// =============================================================================
// 段 9: 合成 PID 目标位置并限位 → 调用 El_Ctrl_FB
// rPIDCmdPos = 程引插值 + 手动偏置 + 自跟踪偏置 + AGC搜索偏置 + 安全检查偏置
// =============================================================================
Axis1Remote.rPIDCmdPos:=RealTimePosCal.rInterElPos+rStepBias+rAuToStepBias+rSearchNextStepTarget+SECURITYCHECK.el_out+rAuToStepBiasTemp;
IF Axis1Remote.rPIDCmdPos<93 THEN
	Axis1Remote.rPIDCmdPos:=93;
ELSIF Axis1Remote.rPIDCmdPos>180 THEN
	Axis1Remote.rPIDCmdPos:=180;
END_IF

Axis1_Ctrl(sLocal:=Axis1Local, sCtrl:=Axis1Remote, sStatus:=Axis1Status, sVisible:=Axis1Visible, rRealPos:=rFctPosReal_1, rPosLimK:=0.34);

                  
END_PROGRAM

FUNCTION_BLOCK LinearInter
  VAR_INPUT
    tLastTime : ULINT;  (* 上一时间 *)
    rLastPos : REAL;  (* 上一时间位置 *)
    tCurTime : ULINT;  (* 当前时间 *)
    rCurPos : REAL;  (* 当前时间位置 *)
    tTargetTime : ULINT;  (* 目标时间 *)
  END_VAR
  VAR_OUTPUT
    rTargetpos : REAL;  (* 目标时间位置 *)
  END_VAR
  VAR
    iDelCurLastTime : LREAL := 1.0;  (* 当前与上一个时间差 *)
    iDelTarCurTime : LREAL := 1.0;  (* 目标与当前时间差 *)
    rK : REAL;  (* 方位斜率 *)
  END_VAR

                    //tLastTime:=tLastTime/1000000;
//tCurTime:=tCurTime/1000000;
//tTargetTime:=tTargetTime/1000000;
iDelTarCurTime:=ULINT_TO_LREAL(tTargetTime)-ULINT_TO_LREAL(tCurTime); //x1-x
IF (tCurTime-tLastTime)<>0 THEN
	iDelCurLastTime:=ULINT_TO_LREAL(tCurTime)-ULINT_TO_LREAL(tLastTime);  //x-x0
ELSE
	iDelCurLastTime:=1.0;
END_IF

IF iDelTarCurTime<>0 THEN
	rK:=(rCurPos-rLastPos)/(iDelCurLastTime);
ELSE
	rK:=0;
END_IF
rTargetpos:=rCurPos+rK*iDelTarCurTime;  //y1 + ((y1-y0)/(x1-x0))*(x-x1)
                  
END_FUNCTION_BLOCK

FUNCTION_BLOCK three2
  VAR_INPUT
    X : ARRAY[1..5] OF LREAL;
    Y : ARRAY[1..5] OF LREAL;
    y0 : REAL := 0;
    yn : REAL := 0;  (* y0,yn表示的是S''(x0)=f''(x0)=y0，S''(xn)=f''(xn)=yn,自然边界即条件值为0 *)
  END_VAR
  VAR_OUTPUT
    M : ARRAY[1..5] OF LREAL;
    A : ARRAY[1..5, 1..5] OF LREAL;
    D : ARRAY[1..3, 1..3] OF LREAL;
    g : ARRAY[1..3] OF LREAL;
    h : ARRAY[1..4] OF LREAL;
  END_VAR
  VAR
    n : INT := 5;
    ypie : ARRAY[1..5] OF REAL;
    j : INT;
    i : INT;
    u : ARRAY[1..3] OF REAL;
    n_ : ARRAY[1..3] OF REAL;
    M_ : ARRAY[1..3] OF REAL;
    solve : solvex;
    iCounttest : INT;
    miu : ARRAY[1..4] OF REAL;
  END_VAR

                    //此函数为M值求值函数
//D,h,A,g,M输出量分别为系数矩阵D，插值宽度h，差商表A，g值,M值 
n:=5;
//A(:,1)=Y'
A[1,1]:=Y[1];A[2,1]:=Y[2];A[3,1]:=Y[3];A[4,1]:=Y[4];A[5,1]:=Y[5];

//A(:,1)=Y'
FOR j :=2 TO 5 DO
	FOR i:=j TO 5 DO
		A[i,j]:=(A[i,j-1]- A[i-1,j-1])/(X[i]-X[i-j+1]);
	END_FOR
END_FOR


FOR i:=1 TO (n-1) DO
	h[i]:=X[i+1]-X[i];
END_FOR


//h[1]:=X[2]-X[1];h[2]:=X[3]-X[2];h[3]:=X[4]-X[3];h[4]:=X[5]-X[4];



//D[1,1]:=2;D[2,2]:=2;D[3,3]:=2;

FOR i:=1 TO n-2 DO
	D[i,i]:=2; 
	IF i=1 THEN
		g[i]:=(6/(h[i+1]+h[i]))*(A[i+2,2]-A[i+1,2])-h[i]/(h[i]+h[i+1])*y0;
	ELSIF i=(n-2) THEN
		g[i]:=(6/(h[i+1]+h[i]))*(A[i+2,2]-A[i+1,2])-(1-h[i]/(h[i]+h[i+1]))*yn;
	ELSE
		g[i]:=(6/(h[i+1]+h[i]))*(A[i+2,2]-A[i+1,2]);
	END_IF
END_FOR



FOR i:=2 TO (n-2) DO
	u[i]:=h[i]/(h[i]+h[i+1]);
	n_[i-1]:=h[i]/(h[i-1]+h[i]);
	D[i-1,i]:=n_[i-1];
	D[i,i-1]:=u[i];
END_FOR


solve(M:=D,G:=g,X=>M_);
M[1]:=0;M[5]:=0;M[2]:=M_[1];M[3]:=M_[2];M[4]:=M_[3];


                  
END_FUNCTION_BLOCK

FUNCTION_BLOCK threesimple2
  VAR_INPUT
    aUTC_TIME : ARRAY[1..5] OF ULINT;  (* 用于三次样条插值的数据 *)
    aPosCmd : ARRAY[1..5] OF LREAL;  (* 用于三次样条插值的数据 *)
    y0 : REAL;
    yn : REAL;  (* y0,yn表示的是S''(x0)=f''(x0)=y0，S''(xn)=f''(xn)=yn,自然边界即条件值为0 *)
    xt : REAL;  (* 所求目标位置 *)
  END_VAR
  VAR_OUTPUT
    sout : REAL;
    nout : INT;
  END_VAR
  VAR
    Three : three2;
    X : ARRAY[1..5] OF LREAL;
    Y : ARRAY[1..5] OF LREAL;
    M : ARRAY[1..5] OF LREAL;
    A : ARRAY[1..5, 1..5] OF LREAL;
    D : ARRAY[1..3, 1..3] OF LREAL;
    g : ARRAY[1..3] OF LREAL;
    h : ARRAY[1..4] OF LREAL;
    n : INT := 5;
    p1 : ARRAY[1..4] OF REAL;
    p2 : ARRAY[1..4] OF REAL;
    p3 : ARRAY[1..4] OF REAL;
    p4 : ARRAY[1..4] OF REAL;
    i : INT;
  END_VAR

                    FOR i:=1 TO 5 DO
	X[i]:=ULINT_TO_LREAL(aUTC_TIME[i]);
	Y[i]:=aPosCmd[i];
END_FOR


Three(X:=X,Y:=Y,y0:=y0,yn:=yn,D=>D,h=>h,A=>A,g=>g,M=>M);

FOR i:=1 TO (n-1) DO
	p1[i]:=M[i]*(X[i+1]-xt)*(X[i+1]-xt)*(X[i+1]-xt)/(6*h[i]);
	p2[i]:=M[i+1]*(xt-X[i])*(xt-X[i])*(xt-X[i])/(6*h[i]);
	p3[i]:=(A[i,1]-M[i]/6*(h[i])*(h[i]))*(X[i+1]-xt)/h[i];
	p4[i]:=(A[i+1,1]-M[i+1]/6*(h[i])*(h[i]))*(xt-X[i])/h[i];
	
	
END_FOR


FOR i:=1 TO (n-1) DO
	IF (xt<=X[i+1])AND (xt>=X[i]) THEN
		nout:=i;
		sout:=p1[nout]+p2[nout]+p3[nout]+p4[nout]; 
	ELSIF xt>X[5] THEN
		nout:=4;
	ELSIF xt<X[1]THEN
		nout:=1;
	END_IF
END_FOR


//要不要判断插值模块是否有效？
sout:=p1[nout]+p2[nout]+p3[nout]+p4[nout]; 
(*
IF xt>X[5] THEN
	nout:=4;
	sout:=p1[nout]+p2[nout]+p3[nout]+p4[nout]; 
ELSIF xt<X[1] THEN
	nout:=1;
	sout:=p1[nout]+p2[nout]+p3[nout]+p4[nout]; 
END_IF
*)
                  
END_FUNCTION_BLOCK

FUNCTION_BLOCK InterDataProcess
  VAR_INPUT
    ulRealTime : ULINT;  (* 实际时间 单位纳秒 *)
    Arr : ARRAY[1..5] OF ULINT := [9, 0, 1, 5, 4];  (* 创建一个包含5个整数的数组 轨道时间数组 起点 1970-01-01 0:00:00 单位纳秒 *)
  END_VAR
  VAR_OUTPUT
    MaxVal : ULINT;  (* 定义最大值、最小值和循环计数器变量 *)
    MinVal : ULINT;  (* 定义最大值、最小值和循环计数器变量 *)
    MaxIndex : INT;  (* 定义最大值和最小值的索引 *)
    MinIndex : INT;  (* 定义最大值和最小值的索引 *)
    ulInterRealTime : ULINT;  (* 插值使用的时间 *)
  END_VAR
  VAR
    i : INT;
    j : INT;
  END_VAR

                    //该功能块查找到轨道时间数组内最大最小值以及索引位置
//找出最大最小值
MaxVal := 0; // 初始化最大值
MinVal := 0; // 初始化最小值
MaxIndex := 0; // 初始化最大值的索引
MinIndex := 0; // 初始化最小值的索引

FOR i := 1 TO 5 DO
    IF Arr[i] <> 0 THEN
        IF MaxVal = 0 THEN
            MaxVal := Arr[i];
            MaxIndex := i;
        ELSIF Arr[i] > MaxVal THEN
            MaxVal := Arr[i];
            MaxIndex := i;
        END_IF

        IF MinVal = 0 THEN
            MinVal := Arr[i];
            MinIndex := i;
        ELSIF Arr[i] < MinVal THEN
            MinVal := Arr[i];
            MinIndex := i;
        END_IF
    END_IF
END_FOR

// MaxVal 和 MinVal 包含了最大值和最小值，不考虑值为0的元素
// MaxIndex 和 MinIndex 包含了最大值和最小值的索引


//当前时间和最大最小比较 
IF ulRealTime<MinVal*1000000 THEN //小于插值范围 取最小时间
	//
	ulInterRealTime:=MinVal*1000000; //应该修改插值位置 而不是时间
ELSIF ulRealTime>MaxVal*1000000THEN //大于插值范围 取最大时间
	//
	ulInterRealTime:=MaxVal*1000000;//应该修改插值位置 而不是时间
ELSE
	//如果内部有0 则不插值选取最新的数据
	FOR j:=1 TO 5 DO
		IF (Arr[i]=0) AND (j<5) THEN
			ulInterRealTime:=Arr[5];//应该修改插值位置 而不是时间
			MaxIndex:=5;
			EXIT;
		ELSIF (Arr[i]=0) AND (j=5) THEN
			//没有输入数据 需要报错吗？
		END_IF
	END_FOR
	//
END_IF
                  
END_FUNCTION_BLOCK

FUNCTION_BLOCK threesimple2_1
  VAR_INPUT
    XModbusUL : ARRAY[1..10] OF ULINT := [1, 2, 3, 4, 5, 6, 7, 8, 9, 10];  (* 输入的Modbus时间数组 *)
    XModbus : ARRAY[1..10] OF LREAL;
    YModbus : ARRAY[1..10] OF LREAL;  (* 输入的Modbus位置数组 *)
    y0 : REAL;
    yn : REAL;  (* y0,yn表示的是S''(x0)=f''(x0)=y0，S''(xn)=f''(xn)=yn,自然边界即条件值为0 *)
    xt : LREAL;  (* 所求目标位置 *)
  END_VAR
  VAR_OUTPUT
    sout : REAL;
    nout : INT;
    ErrCode : INT;
    bSetZero : BOOL;  (* Modbus序列清零标识符； *)
  END_VAR
  VAR
    Three : three2;
    X : ARRAY[1..5] OF LREAL;
    Y : ARRAY[1..5] OF LREAL;
    M : ARRAY[1..5] OF LREAL;
    A : ARRAY[1..5, 1..5] OF LREAL;
    D : ARRAY[1..3, 1..3] OF LREAL;
    g : ARRAY[1..3] OF LREAL;
    h : ARRAY[1..4] OF LREAL;
    n : INT := 5;
    p1 : ARRAY[1..4] OF REAL;
    p2 : ARRAY[1..4] OF REAL;
    p3 : ARRAY[1..4] OF REAL;
    p4 : ARRAY[1..4] OF REAL;
    i : INT;
    ii : INT;  (* 清空序列 *)
    j : INT;  (* 寻找差值区间的循环变量 *)
    k : INT;  (* 插值区间 *)
    iCountOutMaxRange : INT;
    iCountOutMinRange : INT;
    nn : INT;  (* 格式转换循环遍历 *)
    mm : INT;  (* 查重遍历； *)
  END_VAR

                    FOR nn:=1 TO 10 DO
	//XModbus[nn]:=ULINT_TO_LREAL(XModbusUL[nn])*1000000/1000.0;
	XModbus[nn]:=ULINT_TO_LREAL(XModbusUL[nn]-XModbusUL[1])+1.0;
END_FOR
	xt:=xt-ULINT_TO_LREAL(XModbusUL[1])+1.0;
IF ErrCode>0 THEN
	ErrCode:=0;
END_IF


FOR mm:=2 TO 8 DO
	IF XModbus[mm] = XModbus[mm + 1] THEN
		// 找到相等的两个数，进行线性插值
		XModbus[mm + 1] := (XModbus[mm] + XModbus[mm + 2]) / 2.0;
	END_IF;
END_FOR
IF XModbus[1] = XModbus[2] THEN
	// 找到相等的两个数，进行线性插值
	XModbus[1] := XModbus[2]-(XModbus[3]-XModbus[2]);
END_IF;
IF XModbus[9] = XModbus[10] THEN
	// 找到相等的两个数，进行线性插值
	XModbus[10] := XModbus[9]+(XModbus[9]-XModbus[8]);
END_IF;

IF ErrCode <> 0 THEN
	iCountOutMaxRange:=0;
	iCountOutMinRange:=0;
END_IF


//在何处清空序列呢
//bSetZero:=FALSE; //默认不清空

IF  XModbus[10]=0 THEN
	//报错
	ErrCode:=107;//序列为空
ELSE
	IF XModbus[10]-XModbus[1]>2000000 THEN
		sout:=YModbus[10];
	ELSE
		IF xt<XModbus[1] THEN
			sout:=YModbus[1];
			//报故障 累计超时报错
			iCountOutMinRange:=iCountOutMinRange+1;
			IF iCountOutMinRange>5000 THEN
				iCountOutMaxRange:=5001;
				//ErrCode:=108;//偏小超时报错
			END_IF
		ELSIF xt>XModbus[10]  THEN
			sout:=YModbus[10];
			//报故障 累计超时报错
			iCountOutMaxRange:=iCountOutMaxRange+1;
			IF iCountOutMaxRange>5000 THEN
				iCountOutMaxRange:=5001;
				//ErrCode:=109;//偏大超时报错
			END_IF
		ELSE //若所求目标位置在Modbus中间
			iCountOutMaxRange:=0;
			iCountOutMinRange:=0;
			//若不满五个点
			IF XModbus[6]=0 THEN
				sout:=XModbus[10];
			ELSE
				//若满五个点
				//寻找当前插值区间
				FOR j:=2 TO 10 DO
					IF xt<XModbus[j] THEN
						k:=j;
						EXIT;
					END_IF
				END_FOR
				
				IF k=2 THEN
					X[1]:=XModbus[k-1];X[2]:=XModbus[k];X[3]:=XModbus[k+1];X[4]:=XModbus[k+2];X[5]:=XModbus[k+3];
					y[1]:=YModbus[k-1];Y[2]:=YModbus[k];Y[3]:=YModbus[k+1];Y[4]:=YModbus[k+2];Y[5]:=YModbus[k+3];
				ELSIF k>2 AND k<=8 THEN
					X[1]:=XModbus[k-2];X[2]:=XModbus[k-1];X[3]:=XModbus[k];X[4]:=XModbus[k+1];X[5]:=XModbus[k+2];
					Y[1]:=YModbus[k-2];Y[2]:=YModbus[k-1];Y[3]:=YModbus[k];Y[4]:=YModbus[k+1];Y[5]:=YModbus[k+2];
				ELSIF k=9 THEN
					X[1]:=XModbus[k-3];X[2]:=XModbus[k-2];X[3]:=XModbus[k-1];X[4]:=XModbus[k];X[5]:=XModbus[k+1];
					Y[1]:=YModbus[k-3];Y[2]:=YModbus[k-2];Y[3]:=YModbus[k-1];Y[4]:=YModbus[k];Y[5]:=YModbus[k+1];
				ELSIF k=10 THEN
					X[1]:=XModbus[k-4];X[2]:=XModbus[k-3];X[3]:=XModbus[k-2];X[4]:=XModbus[k-1];X[5]:=XModbus[k];
					Y[1]:=YModbus[k-4];Y[2]:=YModbus[k-3];Y[3]:=YModbus[k-2];Y[4]:=YModbus[k-1];Y[5]:=YModbus[k];
				END_IF
				
				
				//开始解算
				Three(X:=X,Y:=Y,y0:=y0,yn:=yn,D=>D,h=>h,A=>A,g=>g,M=>M);
				FOR i:=1 TO (n-1) DO
					p1[i]:=M[i]*(X[i+1]-xt)*(X[i+1]-xt)*(X[i+1]-xt)/(6*h[i]);
					p2[i]:=M[i+1]*(xt-X[i])*(xt-X[i])*(xt-X[i])/(6*h[i]);
					p3[i]:=(A[i,1]-M[i]/6*(h[i])*(h[i]))*(X[i+1]-xt)/h[i];
					p4[i]:=(A[i+1,1]-M[i+1]/6*(h[i])*(h[i]))*(xt-X[i])/h[i];
				END_FOR
				FOR i:=1 TO (n-1) DO
					IF (xt<=X[i+1])AND (xt>=X[i]) THEN
						nout:=i;
						sout:=p1[nout]+p2[nout]+p3[nout]+p4[nout]; 
					ELSIF xt>X[5] THEN
						nout:=4;
					ELSIF xt<X[1]THEN
						nout:=1;
					END_IF
				END_FOR
				sout:=p1[nout]+p2[nout]+p3[nout]+p4[nout]; 
				(*
				IF xt>X[5] THEN
					nout:=4;
					sout:=p1[nout]+p2[nout]+p3[nout]+p4[nout]; 
				ELSIF xt<X[1] THEN
					nout:=1;
					sout:=p1[nout]+p2[nout]+p3[nout]+p4[nout]; 
				END_IF
				*)
				END_IF
			END_IF
			
		END_IF

//修正输入量为长度为10的数组

END_IF	
	




                  
END_FUNCTION_BLOCK

PROGRAM SecurityCheck
  VAR
    bPrelimit_Positive_1 : BOOL;  (* 俯仰预限位-正侧触发（上报 Modbus DI1 B15） *)
    bPrelimit_Negative_1 : BOOL;  (* 俯仰预限位-负侧触发（DI1 B13） *)
    bPrelimit_Positive_2 : BOOL;  (* 方位预限位-正侧（DI1 B11） *)
    bPrelimit_Negative_2 : BOOL;  (* 方位预限位-负侧（DI1 B09） *)
    bPrelimit_1 : BOOL;  (* 俯仰预限位硬件输入汇总（由 IO 映射赋值） *)
    bPrelimit_2 : BOOL;  (* 方位预限位硬件输入汇总 *)
    bFinallimit_1 : BOOL;  (* 俯仰终限位（DI1 B14/B12） *)
    bFinallimit_2 : BOOL;  (* 方位终限位（DI1 B10/B08） *)
    AzError : REAL;  (* 方位跟踪误差 (deg)，供扫描 FB *)
    ElError : REAL;  (* 俯仰跟踪误差 (deg)，供扫描 FB *)
    rELCurrent : REAL;  (* 俯仰伺服电流 (A 或标幺，由驱动换算) *)
    rAzCurrent : REAL;  (* 方位伺服电流 *)
    rTlCurrent : REAL;  (* 倾斜伺服电流 *)
    rAz_realpos : REAL;  (* 方位“安全逻辑用”位置 = -rFctPosReal_2 *)
    rEL_realpos : REAL;  (* 俯仰相对水平仰角 = rFctPosReal_1 - 90 *)
    fbScan : SpiralScan;  (* 直线/栅格扫描（PersistentVars.bSearchType=FALSE） *)
    fbScan1 : SpiralScan_1;  (* 螺旋扫描（bSearchType=TRUE） *)
    fbScantest : SpiralScan;  (* 测试用（已注释） *)
    enabletest : BOOL;
    aztest : REAL;  (* 测试扫描输出（非搜索时叠加到 rPosCmd） *)
    eltest : REAL;
    enable : BOOL;  (* 扫描 FB 使能：双轴程引且 AGC 达门限且未在跟踪 *)
    delta : REAL;
    n_steps : REAL;
    agc_sim : REAL;
    lock_sim : BOOL;
    cycle_cnt : INT;
    sim_done : BOOL;
    az_out : REAL;  (* 扫描给出的方位修正量 → Az rPIDCmdPos 减去此项 *)
    el_out : REAL;  (* 扫描给出的俯仰修正量 → El rPIDCmdPos 加上此项 *)
    done_out : BOOL;  (* 本轮扫描步完成 *)
    bLockSearch : BOOL;  (* 已锁定（信噪/AGC/误差电压条件满足） *)
    rSearchThre : REAL;
    rSearchThreTemp : REAL;
    bStartTrackTemp : BOOL;  (* ACU 请求自跟踪的边沿锁存 *)
    RiseEdge : R_TRIG;  (* Modbus_Slave.bStartTrackAcu 上升沿 *)
    icountLostLocking : INT;  (* 失锁计数（bType_out 路径，约 1000 拍≈10s） *)
    bErrorLock : BOOL;  (* 误差电压小于门限视为“可跟踪” *)
    icountLostLocking1 : INT;  (* 失锁计数（非 bType_out 路径，约 300 拍） *)
    bType_out : BOOL;  (* 扫描 FB 输出：扫描类型/阶段标志 *)
    iconutwait : INT;  (* 扫描完成后等待计数（用于延迟开跟踪） *)
    rdelta : REAL;  (* 螺旋扫描半径步长 *)
    rStep : REAL;  (* 螺旋扫描步数参数 *)
    bFinish : BOOL;  (* 扫描修正后误差足够小（|AzError+az_out|等） *)
    rAzErrorReal : REAL;  (* 滤波误差（已注释） *)
    rElErrorReal : REAL;
    rAlpha : REAL;  (* 滤波系数（已注释） *)
  END_VAR

                    (*==============================================================================
  PRG: SecurityCheck（远控汇总 / 安全联锁 / 捕获扫描 / 自跟踪启停）
  任务: Canopen 10ms（与 *_ctrl_1 同周期，先于或并行执行需注意调用顺序）

  主要职责:
    1. Modbus_Slave → Axis1/2/3Remote 远控命令统一赋值（阶段5 中 *_ctrl_1 注释块已移至此）
    2. 伺服电流监测（%IW10/20/30 × %ID4/9/14）
    3. 俯仰/方位跟踪误差 AzError、ElError（供螺旋/直线扫描 FB）
    4. 预限位 → GVL.Error_code 201/202，状态上报 Modbus DI1
    5. 捕获扫描 SpiralScan：输出 az_out / el_out → 叠加到 rPIDCmdPos
    6. 根据 AGC/锁相/扫描完成 自动置位 GVL.bStartTrack

  与 *_ctrl_1 关系:
    El:  rPIDCmdPos += SecurityCheck.el_out
    Az:  rPIDCmdPos -= SecurityCheck.az_out
==============================================================================*)

// =============================================================================
// 段 1: 安全逻辑用位置（与显示用 rFctPosReal 可能差符号/零点）
// =============================================================================
rAz_realpos := -1 * GVL.rFctPosReal_2;
rEl_realpos := GVL.rFctPosReal_1 - 90;

// =============================================================================
// 段 2: 三轴伺服电流监测（仅使能时读 AD，%IW×%ID/1e6）
// %IW10/%ID4=俯仰, %IW20/%ID9=方位, %IW30/%ID14=倾斜
// =============================================================================
IF Axis1Status.bServo_Enable THEN
	rELCurrent:=DINT_TO_REAL((INT_TO_DINT(%IW10)* %ID4))/1000000.0;  //俯仰轴电流监测
ELSE
	rELCurrent:=0;
END_IF

IF Axis2Status.bServo_Enable THEN
	rAzCurrent:=DINT_TO_REAL((INT_TO_DINT(%IW20)* %ID9))/1000000.0;  //方位轴电流监测
ELSE
	rAzCurrent:=0;
END_IF

IF Axis3Status.bServo_Enable THEN
	rTlCurrent:=DINT_TO_REAL((INT_TO_DINT(%IW30)* %ID14))/1000000.0;  //倾斜轴电流监测
ELSE
	rTlCurrent:=0;
END_IF

// =============================================================================
// 段 3: 跟踪误差（供 SpiralScan 判断扫描方向与完成度）
// mode2 指向: 命令位置 vs 实际位置
// mode4 程引: 插值目标+偏置 vs 实际位置（含手动/自跟踪偏置）
// =============================================================================
IF Axis2Remote.iMode = 2 THEN
	AzError:=(-1) * (Axis2Remote.rPosCmd-rFctPosReal_2);
	ElError:=Axis1Remote.rPosCmd-rFctPosReal_1;	
END_IF

IF Axis2Remote.iMode = 4 THEN
	AzError:=rFctPosReal_2-RealTimePosCal.rInterazPos-(az_ctrl_1.rStepBias+az_ctrl_1.rAuToStepBias);
	ElError:=RealTimePosCal.rInterElPos-rFctPosReal_1+ (El_ctrl_1.rStepBias+EL_ctrl_1.rAuToStepBias);
END_IF
(*
rAzErrorReal := rAzErrorReal + rAlpha * (AzError - rAzErrorReal);
rElErrorReal := rElErrorReal + rAlpha * (ElError - rElErrorReal);
*)

// =============================================================================
// 段 4: 远控故障复位（Modbus bCommReset → GVL.bError_Reset）
// =============================================================================
IF NOT GVL.bLocalCtrl THEN
	IF Modbus_Slave.bCommReset THEN
		GVL.bError_Reset:=TRUE;
	ELSE
		GVL.bError_Reset:=FALSE;
	END_IF
END_IF

// =============================================================================
// 段 5: 远控 rPosCmd 赋值（含 AGC 搜索偏置或测试扫描偏置）
// 非 bSearch: Modbus 目标 + eltest/aztest
// bSearch:   Modbus 目标 + *_ctrl_1 的 rSearchNextStepTarget_tb
// =============================================================================
IF NOT modbus_slave.bSearch THEN
	Axis1Remote.rPosCmd:=Modbus_Slave.rPosCmd_1 + eltest;
	Axis2Remote.rPosCmd:=Modbus_Slave.rPosCmd_2 - aztest;
ELSE
	Axis1Remote.rPosCmd:=Modbus_Slave.rPosCmd_1 + El_ctrl_1.rSearchNextStepTarget_tb;
	Axis2Remote.rPosCmd:=Modbus_Slave.rPosCmd_2 + Az_ctrl_1.rSearchNextStepTarget_tb;
END_IF

// =============================================================================
// 段 6: 远控三轴命令参量 — Modbus_Slave → AxisXRemote（核心汇总）
// 俯仰/方位 rPosCmd 已在段 5 赋值；此处写 mode/速度/PID/加减速等
// =============================================================================
Axis1Remote.iMode:=Modbus_Slave.iMode_1;
Axis1Remote.rVelCmd:=Modbus_Slave.rVelcmd_1;
//Axis1Remote.rPosCmd:=Modbus_Slave.rPosCmd_1;
Axis1Remote.rP:=Modbus_Slave.rP_1;
Axis1Remote.rI:=Modbus_Slave.rI_1;
Axis1Remote.rD:=Modbus_Slave.rD_1;
Axis1Remote.rPIDThre:=Modbus_Slave.rThreshold_1;
Axis1Remote.rAcceleration:=Modbus_Slave.rAcceleration_1;
Axis1Remote.rDeceleration:=Modbus_Slave.rDeceleration_1;
Axis1Remote.rVel_Limit:=Modbus_Slave.rVelLim_1;

Axis2Remote.iMode:=Modbus_Slave.iMode_2;
Axis2Remote.rVelCmd:=Modbus_Slave.rVelcmd_2;
//Axis2Remote.rPosCmd:=Modbus_Slave.rPosCmd_2;
Axis2Remote.rP:=Modbus_Slave.rP_2;
Axis2Remote.rI:=Modbus_Slave.rI_2;
Axis2Remote.rD:=Modbus_Slave.rD_2;
Axis2Remote.rPIDThre:=Modbus_Slave.rThreshold_2;
Axis2Remote.rAcceleration:=Modbus_Slave.rAcceleration_2;
Axis2Remote.rDeceleration:=Modbus_Slave.rDeceleration_2;
Axis2Remote.rVel_Limit:=Modbus_Slave.rVelLim_2;

Axis3Remote.iMode:=Modbus_Slave.iMode_3;
Axis3Remote.rVelCmd:=Modbus_Slave.rVelcmd_3;
Axis3Remote.rPosCmd:=Modbus_Slave.rPosCmd_3;
Axis3Remote.rP:=Modbus_Slave.rP_3;
Axis3Remote.rI:=Modbus_Slave.rI_3;
Axis3Remote.rD:=Modbus_Slave.rD_3;
Axis3Remote.rPIDThre:=Modbus_Slave.rThreshold_3;
Axis3Remote.rAcceleration:=Modbus_Slave.rAcceleration_3;
Axis3Remote.rDeceleration:=Modbus_Slave.rDeceleration_3;

(* 本控 HMI 赋值块已注释，本控参数由其他 POU 写入 AxisXLocal *)

// =============================================================================
// 段 7: 俯仰预限位 → Error_code 201(正)/202(负)，置位上报标志
// bPrelimit_1 由硬件 IO 映射；触发后根据当前位置方向区分正负限位
// =============================================================================
IF bPrelimit_1 THEN
	IF rFctPosReal_1>0 THEN
		bPrelimit_Positive_1:=TRUE;
		Error_code:=201;
	ELSE
		bPrelimit_Negative_1:=TRUE;
		Error_code:=202;
	END_IF;
ELSE
	bPrelimit_Negative_1:=FALSE;
	bPrelimit_Positive_1:=FALSE;
	;
END_IF

// =============================================================================
// 段 8: 方位预限位（仅置标志，Error_code 203/204 已注释）
// =============================================================================
IF bPrelimit_2 THEN
	IF rFctPosReal_2>0 THEN
		//Error_code:=203;
		bPrelimit_Positive_2:=TRUE;;
	ELSE
		//Error_code:=204;
		bPrelimit_Negative_2:=TRUE;;
	END_IF;
ELSE
	bPrelimit_Negative_2:=FALSE;
	bPrelimit_Positive_2:=FALSE;
	;
END_IF

// =============================================================================
// 段 9: 锁定判定 — 信噪比 EB_N0≥28 或 (AGC≥门限 且 误差电压≤rErrorThre)
// bErrorLock: 仅误差电压小（适合进入跟踪）
// =============================================================================
bLockSearch := READ_485.Chan1EB_N0 >= 28 OR ((GVL.Chan1AGC >= GVL.Chanthreshold) AND (SQRT(GVL.Chan1Ua * GVL.Chan1Ua + GVL.Chan1Ue * GVL.Chan1Ue) <= PersistentVars.rErrorThre));
bErrorLock  := (SQRT(GVL.Chan1Ua * GVL.Chan1Ua + GVL.Chan1Ue * GVL.Chan1Ue) <= PersistentVars.rErrorThre);

// =============================================================================
// 段 10: 捕获扫描使能 — 双轴均为程引(4)、AGC 达标或接收机锁定、且尚未自跟踪
// =============================================================================
IF Axis1Remote.iMode = 4 AND Axis2Remote.iMode = 4 AND (gvl.Chan1AGC > PersistentVars.rStartThre OR READ_485.recBuf[1] = 1) AND NOT GVL.bStartTrack THEN
	enable := TRUE;
ELSIF Axis1Remote.iMode <> 4 THEN
	enable := FALSE;
END_IF

// =============================================================================
// 段 11: 调用扫描 FB — 直线(SpiralScan) 或 螺旋(SpiralScan_1)
// 输出 az_out / el_out 在 *_ctrl_1 中叠加到 rPIDCmdPos
// =============================================================================
IF NOT PersistentVars.bSearchType THEN
	// ===== 调用直线扫描 =====
	fbScan(
		enable      := enable,
		delta       := PersistentVars.rAzScanRange,
		delta1      := PersistentVars.rElScanRange,
		n_steps     := PersistentVars.rStep,
		agc      := GVL.Chan1AGC,
		locked     := bLockSearch,
		AzError := AzError,
		elError := elError,
		bTrackState := GVL.bStartTrack,
		azimuth     => az_out,
		elevation   => el_out,
		done        => done_out,
		bType  =>bType_out
	);
ELSE
	// ===== 调用螺旋扫描====
	fbScan1(
		enable      := enable,
		delta       := rdelta,
		n_steps     := rStep,
		agc      := GVL.Chan1AGC,
		locked     := bLockSearch,
		AzError := AzError,
		elError := elError,
		azimuth     => az_out,
		elevation   => el_out,
		done        => done_out,
		bType  =>bType_out
	);
END_IF

// =============================================================================
// 段 12: 自跟踪启停状态机（仅双轴程引 mode4）
// 扫描完成+锁定 → 置 GVL.bStartTrack
// 失锁持续计数超阈值 → 清 GVL.bStartTrack
// PersistentVars.bTrackingMode: TRUE=自动开跟踪, FALSE=需 ACU 边沿 bStartTrackAcu
// =============================================================================
IF Axis1Remote.iMode = 4 AND Axis2Remote.iMode = 4 THEN
	bFinish := done_out AND (ABS(AzError + az_out) <= 0.08) AND (ABS(ElError + el_out) <= 0.08);//扫描到位
	// 上升沿检测
	RiseEdge(CLK := Modbus_Slave.bStartTrackAcu);
	
	IF RiseEdge.Q THEN
		bStartTrackTemp := TRUE;
	END_IF;
	
	IF PersistentVars.bTrackingMode THEN
		IF bType_out THEN
			IF done_out AND bLockSearch THEN
				GVL.bStartTrack := TRUE;
				icountLostLocking := 0;
			ELSIF done_out AND NOT (SQRT(GVL.Chan1Ua * GVL.Chan1Ua + GVL.Chan1Ue * GVL.Chan1Ue) <= PersistentVars.rErrorThre) THEN
				icountLostLocking := icountLostLocking + 1;
				IF icountLostLocking >= 1000 THEN //失锁持续5秒退出自跟踪
					icountLostLocking := 1001;
					GVL.bStartTrack := FALSE;
				END_IF
			END_IF
		ELSE
			IF done_out THEN
				iconutwait := iconutwait + 1;
			END_IF
			IF iconutwait >= 500 THEN
				Iconutwait := 501;
			END_IF
			IF iconutwait >= 100 AND bErrorLock AND (bFinish OR iconutwait >= 500) THEN
				GVL.bStartTrack := TRUE;
				icountLostLocking1 := 0;
			ELSIF iconutwait >= 100 AND NOT bErrorLock THEN
				icountLostLocking1 := icountLostLocking1 + 1;
				IF icountLostLocking1 >= 300 THEN //失锁持续5秒退出自跟踪
					icountLostLocking1 := 301;
					GVL.bStartTrack := FALSE;
				END_IF
			END_IF
		END_IF
	ELSE
		IF bType_out THEN
			IF done_out AND bLockSearch THEN
				GVL.bStartTrack := bStartTrackTemp;
				icountLostLocking := 0;
			ELSIF done_out AND NOT (SQRT(GVL.Chan1Ua * GVL.Chan1Ua + GVL.Chan1Ue * GVL.Chan1Ue) <= PersistentVars.rErrorThre) THEN
				icountLostLocking := icountLostLocking + 1;
				IF icountLostLocking >= 1000 THEN //失锁持续5秒退出自跟踪
					icountLostLocking := 1001;
					GVL.bStartTrack := FALSE;
				END_IF
			END_IF
		ELSE
			IF done_out THEN
				iconutwait := iconutwait + 1;
			END_IF
			IF iconutwait >= 500 THEN
				Iconutwait := 501;
			END_IF
			IF iconutwait >= 100 AND bErrorLock AND (bFinish OR iconutwait >= 500) THEN
				GVL.bStartTrack := bStartTrackTemp;
				icountLostLocking1 := 0;
			ELSIF iconutwait >= 100 AND NOT bErrorLock THEN
				icountLostLocking1 := icountLostLocking1 + 1;
				IF icountLostLocking1 >= 300 THEN //失锁持续5秒退出自跟踪
					icountLostLocking1 := 301;
					GVL.bStartTrack := FALSE;
				END_IF
			END_IF
		END_IF
	END_IF
ELSE
	bStartTrackTemp := FALSE;
	GVL.bStartTrack := Modbus_Slave.bStartTrackAcu;
	icountLostLocking := 0;
	icountLostLocking1 := 0;
	Iconutwait := 0;
END_IF

(* fbScantest 测试块已注释 *)

                  
END_PROGRAM

FUNCTION_BLOCK PID_1
  VAR_INPUT
    rTarget : REAL;  (* 设定值 *)
    rFeedback : REAL;  (* 反馈值 *)
    rPosLimPositive : LREAL;  (* 位置正限位 *)
    rPosLimNegative : LREAL;  (* 位置反限位 *)
    rKp : REAL;  (* 比例增益 *)
    rKi : REAL;  (* 积分增益 *)
    rKd : REAL;  (* 微分增益 *)
    iThreshold : INT;  (* 积分项开启的位置阈值 *)
    bPIDEnable : BOOL := TRUE;  (* PID使能 *)
    rVelLim : LREAL;  (* 速度限制 *)
  END_VAR
  VAR_OUTPUT
    rPIDOutput : LREAL := 0;  (* 带方向的输出速度 *)
  END_VAR
  VAR
    rLastError : LREAL := 0.0;  (* 上一次误差 *)
    rErrorNow : LREAL := 0.0;  (* 当前误差 *)
    rIntegralNew : LREAL := 0.0;  (* 积分项 *)
    rDerivativeNew : LREAL := 0.0;  (* 微分项 *)
    rDelta : LREAL;  (* 增量 *)
    rProportionNew : LREAL;
  END_VAR

                    
IF (bPIDEnable>0) THEN //如果PID使能
	IF rTarget=rFeedback THEN
		rPIDOutput:=0;	
	ELSE
	
		rErrorNow:=rTarget-rFeedback;//计算当前误差 en
		rProportionNew:=rErrorNow;//比例项
		//积分项
		IF rFeedback>rPosLimNegative AND rFeedback<rPosLimPositive THEN //若在软限位之内，工作时开启积分项
			IF (ABS(rTarget-rFeedback)<iThreshold OR iThreshold = -1) THEN//位置差小于积分阈值开始积分，或者设置阈值为-1，不启用这个控制
				rIntegralNew:= rIntegralNew+rErrorNow; //积分项
			ELSE
				rIntegralNew:=0;
			END_IF;
		ELSE //不在软限位范围内,则积分项为0
			rIntegralNew:=0;
		END_IF

		//PID输出
		rPIDOutPut:=rKp*rProportionNew+rKi*rIntegralNew;


		//PID限速
		
			IF rPIDOutput<(-rVelLim) THEN
				rPIDOutput:=-rVelLim;
			ELSIF rPIDOutput>rVelLim THEN
				rPIDOutput:=rVelLim;
			END_IF
		
		
		IF rFeedback>rPosLimPositive AND rPIDOutput>0 THEN 
			rPIDOutput:=0;
		END_IF
		IF rFeedback<rPosLimNegative AND rPIDOutput<0 THEN
			rPIDOutput:=0;
		END_IF
		
		rLastError:=rErrorNow;//将当前误差赋值给上一次误差
		
	END_IF
ELSE//非使能清零PID各项
	rProportionNew:=0.0;
	rIntegralNew:=0.0;
	rPIDOutput:=0.0;
END_IF










                  
END_FUNCTION_BLOCK

PROGRAM AutoTrackingCal
  VAR
    rChanUa : REAL;  (* 处理后方位误差 (V)，→ Az 自跟踪 *)
    rChanUe : REAL;  (* 处理后俯仰误差 (V)，→ El 自跟踪 *)
    rChanAGC : REAL;  (* 当前通道 AGC *)
    bChanLock : BOOL;  (* 通道锁定（保留） *)
    iCountATLock : INT;
    iState : INT;  (* 跟踪通道选择：1=通道1, 2=通道2 *)
    rAzSum : LREAL;  (* 方位累积拉偏 *)
    rElSum : LREAL;  (* 俯仰累积拉偏 *)
    rDirSenFac : REAL;  (* 方向灵敏度系数（除数） *)
    rCurentEl : LREAL;  (* 当前俯仰角弧度 (rFctPosReal_1-90) *)
    rk : LREAL;  (* 累积增益（用于 rAzSum/rElSum） *)
    rChanUaLocal : REAL;  (* 本控方位误差（未见赋值逻辑） *)
    rChanUeLocal : REAL;  (* 本控俯仰误差（未见赋值逻辑） *)
  END_VAR

                    

(*==============================================================================
  PRG: AutoTrackingCal（自跟踪误差电压处理）
  任务: Canopen 10ms
  输入: GVL.Chan1Ua/Ue/AGC/Lock（由 READ_485 写入）
  输出（程序内变量，供 *_ctrl_1 引用）:
    rChanUa  — 方位误差电压（已÷灵敏度、÷cos(俯仰)）
    rChanUe  — 俯仰误差电压（已÷灵敏度）
    rAzSum / rElSum — 累积拉偏量（当前未回写到 GVL）
  使用:
    El_ctrl_1: rChanUe → rChanU / rAuToStepBias
    Az_ctrl_1: -rChanUa → rChanU / rAuToStepBias
  注意:
    rDirSenFac、rk 在导出代码中未见赋值，可能来自 Modbus/HMI 或需人工确认
    rChanUaLocal / rChanUeLocal 未见赋值，本控自跟踪可能依赖未初始化值（原工程保留）
==============================================================================*)
(* 旧版按 iState 直接映射 GVL 通道，已注释 *)

//iState:=modbusSlave.Trace_Num;//跟踪支路选择
iState:=1;                             // 固定使用跟踪接收机 1

CASE iState OF 
	1://使用跟踪接收机1 且锁定标识为True
		// ----- 自跟踪使能且（锁定或 SecurityCheck 误差电压足够小）-----
		IF GVL.bStartTrack AND (GVL.Chan1Lock OR Securitycheck.bErrorLock) THEN
			// 方位：原始 Ua → ÷灵敏度 → ÷cos(El) 补偿大仰角时方位耦合
			rChanUa:=GVL.Chan1Ua;
			rChanUa:=rChanUa/rDirSenFac;
			rCurentEl:=(rFctPosReal_1-90)*3.1415926535897/180.0;
			rChanUa:=rChanUa/COS(rCurentEl);
			
			// 俯仰：原始 Ue → ÷灵敏度
			rChanUe:=GVL.Chan1Ue;
			rChanUe:=rChanUe/rDirSenFac;
			rChanAGC:=GVL.Chan1AGC;
			
			// 累积量（供扩展；当前 *_ctrl_1 主要用瞬时 rChanUa/Ue）
			rAzSum:=rAzSum+rk*rChanUa/1000.0;
			rElSum:=rElSum+rk*rChanUe/1000.0;
		ELSE
			rAzSum:=0;
			rElSum:=0;
			rChanUa:=0;
			rChanUe:=0;
		END_IF
		
	2://使用跟踪接收机2 且锁定标识为True
		rChanUa:=GVL.Chan2Ua;
		rChanUe:=GVL.Chan2Ue;
		rChanAGC:=GVL.Chan2AGC;
		
	3://锁定标识符为False
		//bChanLock:=FALSE;
END_CASE

                  
END_PROGRAM

PROGRAM Ti_ctrl_1
  VAR
    Axis3_Ctrl : Ti_Ctrl_FB;  (* 倾斜轴控制 FB *)
    bRemote2LocalStop : BOOL;
    bLocal2RemoteStop : BOOL;
    Error : INT;
    Axis3Limit_pos : REAL;  (* +190° *)
    Axis3Limit_Neg : REAL;  (* -190° *)
    bRTriger : Standard.R_TRIG;
    bFTriger : Standard.F_TRIG;
    Stop3_Count : INT;
    bStop_3 : BOOL;  (* 倾斜轴停稳标志 *)
    rPosModeStepBias : LREAL;
    rPosModeStep : LREAL;
    rStepBiasMax : LREAL;
    rStepBias : LREAL;
    rStep : LREAL;
    rAuToStepBias : LREAL;
    rAutoStep : LREAL;
    TbAutoTrigger : Standard.F_TRIG;
    RbAutoTrigger : Standard.R_TRIG;
    rAutoTrackingBiasMax : LREAL;
    rLocalInitPosModeSpeed : REAL;
    rRemoteInitPosModeSpeed : REAL;
    iCountOffAuto : INT;
    iCasePBAutoTrack : INT;
    rKAuToStepBias : LREAL;
    bVisError : BOOL;  (* 全局错误可视化 *)
  END_VAR

                    
(*==============================================================================
  PRG: Ti_ctrl_1（倾斜轴 Ti 顶层程序）
  任务: Canopen 10ms
  作用: 倾斜轴反馈、状态、远/本控切换保护，调用 Ti_Ctrl_FB
  与 El/Az 差异:
    - 无 AGC 搜索、无自跟踪拉偏（相关代码已注释）
    - 未在此程序内赋值 rPIDCmdPos（由 Modbus/其他模块写入后仅做限位）
    - 远控→本控切换时仅强制 Axis3Remote.iMode:=7（本控 mode 未同步置 7）
    - 本控上限钳位有一处写 Axis2Local（原工程保留，勿改）
  软限位: ±190°
==============================================================================*)
IF GVL.Error_code <> 0 THEN
	bVisError := TRUE;
ELSE
	bVisError := FALSE;
END_IF

(* 远控参量注释块为历史 Az 轴拷贝，倾斜轴参数由 Modbus_Slave 写入 Axis3Remote *)

// =============================================================================
// 段 1: 驱动状态 → Axis3Status
// =============================================================================
Axis3Status.Error := GVL.bTiStsBit3;
Axis3Status.ErrorID := GVL.eTiErrorcode;
Axis3Status.bServo_Enable := GVL.bTiStsBit0 AND GVL.bTiStsBit1 AND GVL.bTiStsBit2;
Axis3Status.bBrake := NOT (GVL.bTiStsBit0 AND GVL.bTiStsBit1 AND GVL.bTiStsBit2);
Axis3Status.Disabled := NOT (GVL.bTiStsBit0 AND GVL.bTiStsBit1 AND GVL.bTiStsBit2);
Axis3Remote.rSoft_limit_Negative:=-190;Axis3Remote.rSoft_limit_Postive:=190;
Axis3Local.rSoft_limit_Negative:=-190;Axis3Local.rSoft_limit_Postive:=190;

// =============================================================================
// 段 2: CANopen 反馈 → rFctVelReal_3 / rFctPosReal_3
// =============================================================================
rFctVelReal_3:=DINT_TO_REAL(diTiActVel)/524288.0*360.0;
rFctPosReal_3:=DINT_TO_REAL(diTiActPos)/524288.0*360.0;

// =============================================================================
// 段 3: rPosCmd 硬限位 ±190°
// 注意: 上限分支写的是 Axis2Local（原代码），与 Axis3Local 不一致，保持不改
// =============================================================================
Axis3Limit_pos:=190;
Axis3Limit_Neg:=-190;
IF Axis3Remote.rPosCmd>Axis3Limit_pos THEN
	Axis3Remote.rPosCmd:=190;
ELSIF Axis3Remote.rPosCmd<Axis3Limit_Neg THEN
	 Axis3Remote.rPosCmd:=-190;  
END_IF

IF Axis3Local.rPosCmd>Axis3Limit_pos THEN
	Axis2Local.rPosCmd:=190;
ELSIF Axis3Local.rPosCmd<Axis3Limit_Neg THEN
	 Axis3Local.rPosCmd:=-190;  
END_IF

// =============================================================================
// 段 4: 停稳判定 → Axis3Status.Moving
// =============================================================================
IF  ABS(rFctVelReal_3)<0.035 THEN
	Stop3_Count:=Stop3_Count+1;
	IF Stop3_Count>100 THEN
		Stop3_Count:=101;
		bStop_3:=TRUE;;
	END_IF
ELSE
	Stop3_Count:=0;
	bStop_3:=FALSE;
END_IF
Axis3Status.Moving := NOT bStop_3;

// =============================================================================
// 段 5: PID 使能（mode 2 / 4）
// =============================================================================
IF Axis3Remote.iMode=2 OR Axis3Remote.iMode=4 THEN
	Axis3Remote.bPIDEnable:=TRUE;
ELSE
	Axis3Remote.bPIDEnable:=FALSE;
END_IF

// =============================================================================
// 段 6: 远控 ↔ 本控 切换保护
// 远→本: 仅 Axis3Remote.iMode:=7（与 El/Az 双轴同步 halt 不同）
// =============================================================================
bRTriger(CLK:=GVL.bLocalCtrl);
bFTriger(CLK:=GVL.bLocalCtrl);

IF Axis3Status.bServo_Enable AND (bRTriger.Q ) THEN//如果速度不为0且本控发生切换，则减速停止标识为True
	bRemote2LocalStop:=TRUE;
END_IF
IF bRemote2LocalStop  THEN //若减速停止标识符为True 
	
	IF  bStop_3=TRUE THEN//且电机速度不为0 开始减速 减速完成后下使能，下使能完成后复位标识符复位
		Axis3Local.iMode:=0;
		Axis3Remote.iMode:=0;
		IF Axis3Status.bServo_Enable=FALSE THEN
			bRemote2LocalStop:=FALSE;
		END_IF
	ELSE
		Axis3Remote.iMode:=7;
	END_IF
END_IF

IF Axis3Status.bServo_Enable AND (bFTriger.Q ) THEN//如果速度不为0且本控发生切换，则减速停止标识为True
	bLocal2RemoteStop:=TRUE;
END_IF
IF bLocal2RemoteStop  THEN //若减速停止标识符为True 
	
	IF  bStop_3=TRUE THEN//且电机速度不为0 开始减速 减速完成后下使能，下使能完成后复位标识符复位
		Axis3Local.iMode:=0;
		Axis3Remote.iMode:=0;
		IF Axis3Status.bServo_Enable=FALSE THEN
			bLocal2RemoteStop:=FALSE;
		END_IF
	ELSE
		Axis3Remote.iMode:=7;
		Axis3Local.iMode:=7;
	END_IF
END_IF

(* 自跟踪与 rPIDCmdPos 程引合成在此轴已注释，当前仅对既有 rPIDCmdPos 做限位 *)

// =============================================================================
// 段 7: rPIDCmdPos 限位（赋值在其他 POU，如 Modbus_Slave / RealTimePosCal）
// =============================================================================
IF Axis3Remote.rPIDCmdPos<-190 THEN
	Axis3Remote.rPIDCmdPos:=-190;
ELSIF Axis3Remote.rPIDCmdPos>190 THEN
	Axis3Remote.rPIDCmdPos:=190;
END_IF

Axis3_Ctrl(sLocal:=Axis3Local, sCtrl:=Axis3Remote, sStatus:=Axis3Status, sVisible:=Axis3Visible, rRealPos:=rFctPosReal_3, rPosLimK:=0.34);

                  
END_PROGRAM

FUNCTION_BLOCK Ti_Ctrl_FB
  VAR_INPUT
    sLocal : AxisCrtlStruct;  (* 本控命令结构体 *)
    sCtrl : AxisCrtlStruct;  (* 远控命令结构体 *)
    sStatus : AxisStatus;  (* 轴状态 *)
    sVisible : AxisVisible;  (* HMI 可视化（此 FB 未直接使用） *)
    rRealPos : REAL;  (* 编码器实际位置 (deg) *)
    rPosLimK : REAL;  (* 备用限位系数 *)
  END_VAR
  VAR_OUTPUT
    logicError : INT;  (* 保留 *)
  END_VAR
  VAR
    VelPID_1 : PID;  (* positionMode / programBootMode 远控用 *)
    VelPID_2 : PID;  (* 本控 programBootMode 用 *)
    TON_0 : TON;  (* 超时 1s 强制下电计时器 *)
    bTick : BOOL;  (* stop0 超时标志 *)
    tr : BOOL;  (* 心跳恢复进行中标志 *)
    icount1 : INT;  (* 心跳恢复计数器1 *)
    icount2 : INT;  (* 心跳恢复计数器2 *)
    icount3 : INT;  (* 备用 *)
    bfin1 : BOOL;  (* 计数器1完成标志 *)
    bfin2 : BOOL;  (* 保留 *)
    istate : INT;  (* 上电状态机 *)
    icount : INT;  (* 上电步骤计数 *)
  END_VAR

                    (*==============================================================================
  FB: Ti_Ctrl_FB（倾斜轴 Tilt 控制功能块）
  与 El_Ctrl_FB / Az_Ctrl_FB 结构基本相同，主要差异:
    - 操作的 GVL 变量为 Ti 系列（diTiTargetVel / bTiCtrlBitX / eTiErrorcode 等）
    - 无 vpid1（Ti 轴不做变增益，programBootMode 远控直接用 VelPID_1）
    - positionMode 加速度为 10 deg/s²
    - positionMode bStartAutoTrack 分支注释掉（Ti 无自跟踪需求）
    - programBootMode 本控用 VelPID_2，参数直接来自 sLocal.rP/rI/rD
    - programBootMode 远控 bStartAutoTrack=TRUE 时调用 VelPID_1（非 vpid1）

  速度换算公式（通用）:
    diTiTargetVel [inc/s] = deg/s × 524288 / 360
==============================================================================*)

// =============================================================================
// 段 A: 轴停止或下电时清快速停止位 bit8
// =============================================================================
IF sStatus.Disabled OR(NOT sStatus.Moving)THEN
	bTiCtrlBit8 := FALSE;
END_IF

// =============================================================================
// 段 B: 全局错误复位
// =============================================================================
IF GVL.bError_Reset THEN
	sCtrl.iMode:=6;
	sLocal.iMode:=6;
	GVL.Error_code:=0;
END_IF
IF GVL.Error_code =0 THEN
	GVL.bError_Reset:=FALSE;
END_IF

// =============================================================================
// 段 C: CANopen 心跳超时（0x8130）自动恢复序列
// =============================================================================
IF GVL.eTiErrorcode = 16#8130 AND NOT tr THEN
	GVL.bTiCtrlBit7 := TRUE;
	tr:=TRUE;
	istate:=0;
	icount:=0;
	// 写入下电控制字
	GVL.bTiCtrlBit3 := FALSE;
	GVL.bTiCtrlBit0 := FALSE;
	GVL.bTiCtrlBit1 := FALSE;
	GVL.bTiCtrlBit2 := FALSE;
END_IF
IF tr THEN
	icount1 := icount1 + 1;
END_IF
IF icount1 > 101 THEN
	icount1 := 0;
	tr := FALSE;
	GVL.bTiCtrlBit7 := FALSE;
	bfin1 := TRUE;
END_IF
IF bfin1 THEN
	icount2 := icount2 + 1;
END_IF
IF icount2 > 101 THEN
	bfin1 := FALSE;
	icount2 := 0;
END_IF

// =============================================================================
// 段 D: 主控制逻辑
// =============================================================================
IF GVL.Error_code=0 AND GVL.eTiErrorcode = 0 AND NOT GVL.bTiCtrlBit7  AND NOT tr AND NOT bfin1 AND NOT bfin2 THEN

	// =========== 远控 ===========
	IF GVL.bLocalCtrl=FALSE THEN //远控
		IF sCtrl.iMode <> 1 THEN
			istate:=0;
			icount:=0;
		END_IF
		CASE sCtrl.iMode OF

			MODES.powerOff: // 下电
				IF NOT sStatus.Disabled THEN
					IF sStatus.Moving THEN // 运动中，先停止运动
						GVL.diTiTargetVel := 0;
						bTiCtrlBit8 := TRUE;
					ELSE
						// 写入下电控制字
						GVL.bTiCtrlBit3 := FALSE;
						GVL.bTiCtrlBit0 := FALSE;
						GVL.bTiCtrlBit1 := FALSE;
						GVL.bTiCtrlBit2 := FALSE;
					END_IF
				END_IF

			MODES.powerOn:  // 上电（DS402 三步序列）
				IF sStatus.Disabled THEN
					GVL.diTiTargetVel := 0;
					IF GVL.siTiMode <> 3 THEN // 上电时模式默认为3，速度模式
						GVL.siTiMode := 3;
					END_IF
					IF siTiMode = 3 THEN
						CASE istate OF
							0:
								GVL.bTiCtrlBit1 := TRUE;
								GVL.bTiCtrlBit2 := TRUE;
								icount := icount + 1;
								IF icount = 20 THEN
									icount:=0;
									istate:=1;
								END_IF
							1:
								GVL.bTiCtrlBit0 := TRUE;
								icount := icount + 1;
								IF icount = 20 THEN
									icount:=0;
									istate:=2;
								END_IF
							2:
								GVL.bTiCtrlBit3 := TRUE;
						END_CASE
					END_IF
				ELSE
					IF sStatus.Moving THEN
						GVL.diTiTargetVel := 0;
						bTiCtrlBit8 := TRUE;
					ELSE
						bTiCtrlBit8 := FALSE;
					END_IF
				END_IF

			MODES.positionMode: // 远控指向模式（加速度 10 deg/s²，Kp=0.8）
				IF NOT sStatus.Disabled THEN
					IF sCtrl.bStartAutoTrack THEN
						// Ti 轴自跟踪分支已注释掉，实际走 ELSE
						(*
						VelPID_1(rTarget:=sCtrl.rChanU + rRealPos,
								rFeedback:=rRealPos,
								rPosLimPositive:=sCtrl.rSoft_limit_Postive,
								rPosLimNegative:=sCtrl.rSoft_limit_Negative,
								rVelLim:=sCtrl.rVel_Limit,
								rKp:=sCtrl.rP_AutoTrack,//自跟踪PI系数3,0.02
								rKi:=sCtrl.rI_AutoTrack,
								rKd:=sCtrl.rD,
								bPIDEnable:=sCtrl.bPIDEnable,
								iThreshold:= -1,
								rPIDOutput=>sCtrl.rPIDCmdVel);
*)							
					ELSE
						//PID计算速度指令
						VelPID_1(rTarget:=sCtrl.rPosCmd,
							rFeedback:=rRealPos,
							rVelLim:=sCtrl.Pos_Vel,
							rPosLimPositive:=sCtrl.rSoft_limit_Postive,
							rPosLimNegative:=sCtrl.rSoft_limit_Negative,
							rKp:=0.8,//程引PI系数地带：1,0.002  高带：3,0.02
							rKi:=0,
							rKd:=0,
							bPIDEnable:=sCtrl.bPIDEnable,
							iThreshold:=sCtrl.rPIDThre,
							rPIDOutput=>sCtrl.rPIDCmdVel);
					END_IF
					GVL.diTiTargetVel := REAL_TO_DINT(sCtrl.rPIDCmdVel * 524288 / 360);
					GVL.diTiTargetAcc := REAL_TO_UDINT(10 * 524288 / 360);   //加速度 10 deg/s²
					GVL.diTiTargetDec := REAL_TO_UDINT(10 * 524288 / 360);   //减速度
				END_IF

			MODES.velocityMode://手控速度模式-远控模式
				IF NOT sStatus.Disabled THEN
					IF ABS(sCtrl.rVelCmd) <= sCtrl.rVel_Limit THEN
						GVL.diTiTargetVel := REAL_TO_DINT(sCtrl.rVelCmd * 524288 / 360);
					ELSIF sCtrl.rVelCmd > sCtrl.rVel_Limit THEN
						GVL.diTiTargetVel := REAL_TO_DINT(sCtrl.rVel_Limit * 524288 / 360);
					ELSE
						GVL.diTiTargetVel := REAL_TO_DINT(-sCtrl.rVel_Limit * 524288 / 360);
					END_IF
					GVL.diTiTargetAcc := REAL_TO_UDINT(sCtrl.rAcceleration * 524288 / 360);   //加速度
					GVL.diTiTargetDec := REAL_TO_UDINT(sCtrl.rDeceleration * 524288 / 360);   //减速度
				END_IF

			MODES.programBootMode://PID速度模式-正常模式 程引（Ti 轴用 VelPID_1，非 vpid）
				IF NOT sStatus.Disabled THEN
					IF sCtrl.bStartAutoTrack THEN
						// 程引+自跟踪：误差电压叠加到插值位置
						VelPID_1(rTarget:=sCtrl.rChanU + rRealPos,
								rFeedback:=rRealPos,
								rPosLimPositive:=sCtrl.rSoft_limit_Postive,
								rPosLimNegative:=sCtrl.rSoft_limit_Negative,
								rVelLim:=sCtrl.rVel_Limit,
								rKp:=sCtrl.rP_AutoTrack,//自跟踪PI系数3,0.02
								rKi:=sCtrl.rI_AutoTrack,
								rKd:=sCtrl.rD,
								bPIDEnable:=sCtrl.bPIDEnable,
								iThreshold:= -1,
								rPIDOutput=>sCtrl.rPIDCmdVel);							
					ELSE
						//PID计算速度指令（参数来自 sCtrl.rP/rI/rD，由 Modbus/上位机配置）
						VelPID_1(rTarget:=sCtrl.rPIDCmdPos,
							rFeedback:=rRealPos,
							rVelLim:=sCtrl.rVel_Limit,
							rPosLimPositive:=sCtrl.rSoft_limit_Postive,
							rPosLimNegative:=sCtrl.rSoft_limit_Negative,
							rKp:=sCtrl.rP,//程引PI系数地带：1,0.002  高带：3,0.02
							rKi:=sCtrl.rI,
							rKd:=sCtrl.rD,
							bPIDEnable:=sCtrl.bPIDEnable,
							iThreshold:=sCtrl.rPIDThre,
							rPIDOutput=>sCtrl.rPIDCmdVel);
					END_IF
					GVL.diTiTargetVel := REAL_TO_DINT(sCtrl.rPIDCmdVel * 524288 / 360);
					GVL.diTiTargetAcc := REAL_TO_UDINT(sCtrl.rAcceleration * 524288 / 360);   //加速度
					GVL.diTiTargetDec := REAL_TO_UDINT(sCtrl.rDeceleration * 524288 / 360);   //减速度
				END_IF

			MODES.reset://重置
				IF NOT sStatus.Disabled THEN
					IF sStatus.Moving THEN
						GVL.diTiTargetVel := 0;
						bTiCtrlBit8 := TRUE;
					ELSE
						bTiCtrlBit8 := FALSE;
					END_IF
				END_IF

			MODES.halt://待机
				IF NOT sStatus.Disabled THEN
					IF sStatus.Moving THEN
						GVL.diTiTargetVel := 0;
						bTiCtrlBit8 := TRUE;
					ELSE
						bTiCtrlBit8 := FALSE;
					END_IF
				END_IF
			
		END_CASE

	// =========== 本控 ===========
	ELSE // 本控
		IF sLocal.iMode <> 1 THEN
			istate:=0;
			icount:=0;
		END_IF
		CASE sLocal.iMode OF

			MODES.powerOff: // 下电
				IF NOT sStatus.Disabled THEN
					IF sStatus.Moving THEN // 运动中，先停止运动
						GVL.diTiTargetVel := 0;
						bTiCtrlBit8 := TRUE;
					ELSE
						// 写入下电控制字
						GVL.bTiCtrlBit3 := FALSE;
						GVL.bTiCtrlBit0 := FALSE;
						GVL.bTiCtrlBit1 := FALSE;
						GVL.bTiCtrlBit2 := FALSE;
					END_IF
				END_IF

			MODES.powerOn:  // 上电
				IF sStatus.Disabled THEN
					GVL.diTiTargetVel := 0;
					IF GVL.siTiMode <> 3 THEN // 上电时模式默认为3，速度模式
						GVL.siTiMode := 3;
					END_IF
					IF siTiMode = 3 THEN
						CASE istate OF
							0:
								GVL.bTiCtrlBit1 := TRUE;
								GVL.bTiCtrlBit2 := TRUE;
								icount := icount + 1;
								IF icount = 20 THEN
									icount:=0;
									istate:=1;
								END_IF
							1:
								GVL.bTiCtrlBit0 := TRUE;
								icount := icount + 1;
								IF icount = 20 THEN
									icount:=0;
									istate:=2;
								END_IF
							2:
								GVL.bTiCtrlBit3 := TRUE;
						END_CASE
					END_IF
				ELSE
					IF sStatus.Moving THEN
						GVL.diTiTargetVel := 0;
						bTiCtrlBit8 := TRUE;
					ELSE
						bTiCtrlBit8 := FALSE;
					END_IF
				END_IF

			MODES.velocityMode://手控速度模式-本控模式
				IF NOT sStatus.Disabled THEN
					IF ABS(sLocal.rVelCmd) <= sLocal.rVel_Limit THEN
						GVL.diTiTargetVel := REAL_TO_DINT(sLocal.rVelCmd * 524288 / 360);
					ELSIF sLocal.rVelCmd > sLocal.rVel_Limit THEN
						GVL.diTiTargetVel := REAL_TO_DINT(sLocal.rVel_Limit * 524288 / 360);
					ELSE
						GVL.diTiTargetVel := REAL_TO_DINT(-sLocal.rVel_Limit * 524288 / 360);
					END_IF
					GVL.diTiTargetAcc := REAL_TO_UDINT(sLocal.rAcceleration * 524288 / 360);   //加速度
					GVL.diTiTargetDec := REAL_TO_UDINT(sLocal.rDeceleration * 524288 / 360);   //减速度
				END_IF

			MODES.programBootMode://本控位置模式（普通 PID，参数来自 sLocal.rP/rI/rD）
				IF NOT sStatus.Disabled THEN
					IF NOT sLocal.bPIDEnable THEN
						GVL.diTiTargetVel := 0;							
					ELSE
						//PID计算速度指令
						 VelPID_2(rTarget:=sLocal.rPosCmd,
							     rFeedback:=rRealPos,
								 rPosLimPositive:=sLocal.rSoft_limit_Postive,//软限位
								 rPosLimNegative:=sLocal.rSoft_limit_Negative,
								 rKp:=sLocal.rP,
								 rKi:=sLocal.rI,
								 rKd:=sLocal.rD,
								 iThreshold:=sLocal.rPIDThre,
								 bPIDEnable:=sLocal.bPIDEnable,
								 rVelLim:=sLocal.Pos_Vel,
								 rPIDOutput=>sLocal.rPIDCmdVel);//普通PID
					END_IF
					GVL.diTiTargetVel := REAL_TO_DINT(sLocal.rPIDCmdVel * 524288 / 360);
					GVL.diTiTargetAcc := REAL_TO_UDINT(sLocal.rAcceleration * 524288 / 360);   //加速度
					GVL.diTiTargetDec := REAL_TO_UDINT(sLocal.rDeceleration * 524288 / 360);   //减速度
				END_IF

			MODES.reset://重置
			// 是否需要
			MODES.halt://待机
				IF NOT sStatus.Disabled THEN
					IF sStatus.Moving THEN
						GVL.diTiTargetVel := 0;
						bTiCtrlBit8 := TRUE;
					ELSE
						bTiCtrlBit8 := FALSE;
					END_IF
				END_IF
			
		END_CASE
	END_IF

// =============================================================================
// 段 E: 全局错误时强制停轴，超时后强制下电
// =============================================================================
ELSIF GVL.Error_code<>0 AND GVL.eTiErrorcode = 0 AND NOT GVL.bTiCtrlBit7  AND NOT tr AND NOT bfin1 AND NOT bfin2 THEN
	// 出现错误，轴停止运动
	GVL.diTiTargetVel := 0;
	bTiCtrlBit8 := TRUE;
	TON_0(IN:=bTiCtrlBit8,PT:=T#1S,Q=>,ET=>);//判断stop0执行是否超时,若超时强制下电（手动复位）
	IF TON_0.Q THEN
		bTick:=TRUE;
	END_IF
	IF bTick AND sStatus.Moving THEN // 超时强制下电
		// 写入下电控制字
		GVL.bTiCtrlBit3 := FALSE;
		GVL.bTiCtrlBit0 := FALSE;
		GVL.bTiCtrlBit1 := FALSE;
		GVL.bTiCtrlBit2 := FALSE;
	END_IF
END_IF

                  
END_FUNCTION_BLOCK

FUNCTION_BLOCK vpid
  VAR_INPUT
    rTarget : REAL;  (* 目标位置 (deg) *)
    rFeedback : REAL;  (* 实际位置 (deg) *)
    rPosLimPositive : LREAL;  (* 软限位正限 (deg) *)
    rPosLimNegitive : LREAL;  (* 软限位负限 (deg)（注：原拼写 Negitive，勿改） *)
    rKpBase : REAL;  (* Kp 基础值（低速/低角度区） *)
    rKiBase : REAL;  (* Ki 基础值 *)
    rVelThreshold : LREAL;  (* 增益切换阈值：rElPos 超过此值开始叠加增益 *)
    rKpScale : REAL;  (* Kp 随角度的线性缩放斜率 *)
    rKiScale : REAL;  (* Ki 随角度的线性缩放斜率 *)
    iThrehold : INT;  (* 积分开启的误差阈值 (deg) *)
    bPIDEnable : BOOL;  (* PID 使能 *)
    rVelLim : LREAL;  (* 输出速度限幅 (deg/s) *)
    rKpMax : REAL;  (* Kp 上限 *)
    rKiMax : REAL;  (* Ki 上限 *)
    rElPos : REAL;  (* 当前俯仰实际角度，用于动态调整增益（GVL.rFctPosReal_1-90） *)
  END_VAR
  VAR_OUTPUT
    rPIDOutput : LREAL;  (* 不带限位检查的原始输出（内部过渡量） *)
    rPIDOutDir : LREAL;  (* 最终输出速度 (deg/s)，写 diXxTargetVel 前换算 *)
  END_VAR
  VAR
    rLastFeedback : LREAL;  (* 备用（当前版本已注释掉速度计算） *)
    rErrorNow : LREAL;  (* 当前位置误差 *)
    rIntegralNew : LREAL;  (* 积分累计 *)
    rDelta : LREAL;  (* 备用 *)
    rProportionNew : LREAL;  (* 比例项 = rErrorNow *)
    rSpeed : REAL;  (* 备用（速度自适应已注释） *)
    rKp : REAL;  (* 当前实际 Kp（动态跟踪 rKpTarget） *)
    rKi : REAL;  (* 当前实际 Ki *)
    rInterValueNow : LREAL;  (* 备用（插值速度，已注释） *)
    rInterValueLast : LREAL;  (* 备用 *)
    rStep : LREAL;  (* Kp/Ki 每拍变化步长（防止突变） *)
    rKpTarget : REAL;  (* 目标 Kp（由 rElPos 计算） *)
    rKiTarget : REAL;  (* 目标 Ki *)
  END_VAR

                    (*==============================================================================
  FB: vpid（变增益自适应 PID）
  任务: Canopen 10ms（由 El_Ctrl_FB / Az_Ctrl_FB 在 programBootMode 下调用）
  作用: 与 PID 相似，但 Kp/Ki 根据当前俯仰角（rElPos）动态调整
        俯仰角越大（天线仰角越高），摩擦力和惯量变化大，需更高增益
  与 PID 的区别:
    - 输入参数带 Kp/Ki 基础值、缩放因子、最大值
    - 内部按 rElPos > rVelThreshold 时线性增加 Kp/Ki
    - 输出走 rPIDOutDir（方向输出）而非 rPIDOutput
  来源参数: PersistentVars.rXxKpBase/rXxKiBase 等（掉电保持，可由 HMI/Modbus 标定）
==============================================================================*)

// ----- 段：PID 使能入口 -----
IF (bPIDEnable) THEN // 如果PID使能
    IF rTarget = rFeedback THEN
        rPIDOutDir := 0;    
    ELSE
        rErrorNow := rTarget - rFeedback; // 计算当前误差
        rProportionNew := rErrorNow;      // 比例项
		
		// ----- 段：根据俯仰角动态计算目标 Kp/Ki -----
		// rElPos = 当前俯仰角 - 90，即相对水平的仰角
		// 当仰角 > rVelThreshold 时，增益线性增加
		IF rElPos > rVelThreshold THEN
			rKpTarget := rKpBase + rKpScale * (rElPos - rVelThreshold);
			rKiTarget := rKiBase + rKiScale * (rElPos - rVelThreshold);
		ELSE
			rKpTarget := rKpBase;
			rKiTarget := rKiBase;
		END_IF
        // ----- 段：Kp/Ki 上限保护 -----
        IF rKpTarget > rKpMax THEN
			rKpTarget := rKpMax;
		END_IF
		IF rKiTarget > rKiMax THEN
			rKiTarget := rKiMax;
		END_IF
		
		// ----- 段：Kp/Ki 平滑追踪目标值（rStep 步进，防增益突变抖动）-----
		IF rKp<=rKpTarget THEN
			rKp:=rKp+rStep;
		ELSE
			rKp:=rKp-rStep;
		END_IF
		IF rKi<=rKiTarget THEN
			rKi:=rKi+(rKiScale/rKpScale)*rStep;
		ELSE
			rKi:=rKi-(rKiScale/rKpScale)*rStep;
		END_IF
	END_IF

        // ----- 段：条件积分（与 PID 相同逻辑）-----
        IF rFeedback > rPosLimNegitive AND rFeedback < rPosLimPositive THEN // 若在软限位之内，工作时开启积分项
            IF (ABS(rTarget - rFeedback) < iThrehold) THEN // 位置差小于积分阈值
                rIntegralNew := rIntegralNew + rErrorNow;  // 积分项
            ELSE
                rIntegralNew := rIntegralNew;  // 积分项
            END_IF;
        ELSE // 不在软限位范围内，则积分项为0
            rIntegralNew := 0;
        END_IF
        (*
        // 防止目标位置与当前位置偏差过大，导致比例项输出太大，引起震动
        IF rKp * rProportionNew > 2 THEN
            rPIDOutput := 2;
        ELSIF rKp * rProportionNew < -2 THEN
            rPIDOutput := -2;
        ELSE
            rPIDOutput := rKp * rProportionNew + rKi * rIntegralNew / 1000.0; // 由于需求积分项过小，因此积分系数在接口数据上除1000
        END_IF
        *)
		rPIDOutput := rKp * rProportionNew + rKi * rIntegralNew; // 由于需求积分项过小，因此积分系数在接口数据上除1000
        // 根据方向设置输出
        IF rPIDOutput < 0 THEN
            rPIDOutDir := rPIDOutput;
        ELSE
            rPIDOutDir := rPIDOutput;
        END_IF
        
        // ----- 段：速度限幅 -----
        IF (ABS(rPIDOutDir) > rVelLim) THEN
            IF rPIDOutDir < (-rVelLim) THEN
                rPIDOutDir := -rVelLim;
            ELSIF rPIDOutDir > rVelLim THEN
                rPIDOutDir := rVelLim;
            END_IF
        END_IF
        
        // ----- 段：超软限位时强制输出清零 -----
        IF rFeedback > rPosLimPositive AND rPIDOutDir > 0  THEN
            rPIDOutDir := 0;
        END_IF
        IF rFeedback < rPosLimNegitive AND rPIDOutDir <= 0 THEN
            rPIDOutDir := 0;
        END_IF
        
        //rLastFeedback := rFeedback; // 将当前反馈值赋值给上一次反馈值
		//rInterValueLast := rInterValueNow; // 将当前插值位置值赋值给上一次

ELSE // 非使能清零PID各项
    rProportionNew := 0.0;
    rIntegralNew := 0.0;
    rPIDOutDir := 0.0;
    rPIDOutput := 0.0;
END_IF

                  
END_FUNCTION_BLOCK

PROGRAM READ_485
  VAR
    com_init : gcan.FB_Com_Init;
    com_read : gcan.FB_Com_Read;
    com_write : gcan.FB_Com_Write;
    m_uiError : UINT;
    m_out : BOOL;
    isFirst : BOOL;
    mPort : BYTE;  (* 2 = 485 口 *)
    recSize : UINT;
    recBuf : ARRAY[0..19] OF BYTE;  (* 原始接收缓冲（对外可读 recBuf[1] 等） *)
    recData : ARRAY[0..8] OF BYTE;  (* 旧协议 0x7E 帧解析用（已注释） *)
    wAGC : WORD;
    iUa : INT;
    iUe : INT;
    iChan1DataLen : UINT;
    chan1_i : INT;
    chan1_j : INT;
    Word2Bit1 : Word2Bit;  (* AGC 高低字节 → WORD *)
    Word2Bit2 : Word2Bit;  (* Ua → INT *)
    Word2Bit3 : Word2Bit;  (* Ue → INT *)
    rUagcTemp : REAL;
    rUaTemp : REAL;
    rUeTemp : REAL;
    btest : BOOL;
    btest2 : BOOL;
    rSData : REAL;  (* 信号分量（DWORD 差） *)
    rQData : REAL;  (* 噪声分量 *)
    Dword2Bit1 : Dword2Bit;  (* recBuf[8..11] → DWORD *)
    Dword2Bit2 : Dword2Bit;  (* recBuf[12..15] → DWORD *)
    Chan1EB_N0 : REAL;  (* 等效 Eb/N0 (dB)，SecurityCheck.bLockSearch 用 *)
    bEBN0Lock : BOOL;  (* 信噪比锁定标志（与模式/失锁计数相关） *)
    icount0 : INT;  (* recBuf[1]=0 累计，>400 清 bEBN0Lock *)
  END_VAR

                    

(*==============================================================================
  PRG: READ_485（跟踪接收机 RS485 通信）
  任务: SerialCom 5ms（与 GPRMC_1 同任务，端口不同）
  硬件: GCAN 串口 mPort=2（485），19200 8N1
  作用:
    - 读跟踪接收机上报帧 → 解析 AGC、Ua、Ue、锁定、Eb/N0
    - 写入 GVL.Chan1AGC / Chan1Ua / Chan1Ue / Chan1Lock
    - 输出 Chan1EB_N0、recBuf[1]、bEBN0Lock 供 SecurityCheck / 捕获扫描
  帧布局（当前简化协议，非 0x7E 定界）:
    recBuf[1]     — 锁定标志 (1=锁定)
    recBuf[2..3]  — AGC 原始 WORD
    recBuf[4..5]  — 方位误差 Ua 原始 INT
    recBuf[6..7]  — 俯仰误差 Ue 原始 INT
    recBuf[8..15] — Eb/N0 用两路 DWORD 算信噪比
==============================================================================*)

mPort:=2;								//串口端口号设定

// ----- 首次上电：485 初始化 19200 -----
IF isFirst THEN
	com_init(
	EN_IN:=TRUE,
	xEnable:=TRUE,
	bPort:=mPort,
	uiBaudrate:=19200,
	bParity:=0,
	bDatabits:=8,
	bStopbits:=1,
	EN_OUT=>m_out,
	uiError=>m_uiError);
	isfirst:=FALSE;

ELSE
	com_read(
	EN_in:=TRUE,
	bPort:=mPort,
	p_brxdata:=ADR(recBuf),
	uiMaxsize:=20,
	EN_out=>m_out,
	uiRecSize=>recSize,
	uierror=>m_uierror);
	
	// ----- 段 1: 锁定标志 → GVL.Chan1Lock -----
	//GVL.Chan1Lock := BYTE_TO_BOOL(recBuf[1]);
	IF recBuf[1] = 1 AND GVL.Chan1AGC >= GVL.Chanthreshold THEN
		GVL.Chan1Lock := TRUE;
	ELSE
		GVL.Chan1Lock := FALSE;
	END_IF

	// ----- 段 2: 按字节拼接 WORD/INT（Word2Bit UNION）-----
	Word2Bit1.Apart_Byte[1] := recBuf[2];
	Word2Bit1.Apart_Byte[2] := recBuf[3];
	wAGC:=Word2Bit1.Apart_Word;
	
	Word2Bit2.Apart_Byte[1] := recBuf[4];
	Word2Bit2.Apart_Byte[2] := recBuf[5];
	iUa:=Word2Bit2.Apart_INT;
	
	Word2Bit3.Apart_Byte[1] := recBuf[6];
	Word2Bit3.Apart_Byte[2] := recBuf[7];
	iUe:=Word2Bit3.Apart_INT;

	// ----- 段 3: 换算为物理量并限幅后写 GVL -----
	// Ua/Ue: ±5V 满量程对应 INT±2048；AGC: 5 - (raw×5/76) 越大信号越强
	IF ABS(INT_TO_REAL(iUa) * 5 / 2048) <= 5 AND ABS(INT_TO_REAL(iUe) * 5 / 2048) <= 5 AND ABS((WORD_TO_REAL(wAGC) * 5 / 76)) <=5 THEN
		GVL.Chan1Ua := INT_TO_REAL(iUa) * 5 / 2048;
		GVL.Chan1Ue := INT_TO_REAL(iUe) * 5 / 2048;
		GVL.Chan1AGC := 5 - (WORD_TO_REAL(wAGC) * 5 / 76);
	END_IF
	
	// ----- 段 4: Eb/N0 估算（两 DWORD，字节序见 Dword2Bit 填入顺序）-----
	Dword2Bit1.Apart_Byte[3] := recBuf[8];
	Dword2Bit1.Apart_Byte[4] := recBuf[9];
	Dword2Bit1.Apart_Byte[1] := recBuf[10];
	Dword2Bit1.Apart_Byte[2] := recBuf[11];	
	
	Dword2Bit2.Apart_Byte[3] := recBuf[12];
	Dword2Bit2.Apart_Byte[4] := recBuf[13];
	Dword2Bit2.Apart_Byte[1] := recBuf[14];
	Dword2Bit2.Apart_Byte[2] := recBuf[15];	
	
	rQData:=DWORD_TO_REAL(Dword2Bit2.Apart_DWORD);
	rSData:=DWORD_TO_REAL(Dword2Bit1.Apart_DWORD)-rQData;
	
	IF rSData<>0  AND rQData<>0  THEN
		Chan1EB_N0 := 10*LOG(ABS(rSData/rQData))+3.8;
	ELSE
		Chan1EB_N0 := 0;
	END_IF
	
	// ----- 段 5: bEBN0Lock — 程引/指向且 Eb/N0≥29 或 ACU 请求自跟踪 -----
	IF ((GVL.Axis1Remote.iMode = 2 OR GVL.Axis1Remote.iMode = 4) AND Chan1EB_N0 >= 29)AND READ_485.recBuf[1] = 1 OR Modbus_Slave.bStartTrackAcu THEN
		icount0:=0;
		bEBN0Lock := TRUE;
	END_IF
	// 锁定字节为 0 时累计；超 400 拍或下电则清 bEBN0Lock
	IF ( GVL.Axis1Remote.iMode = 4 or GVL.Axis1Remote.iMode =2 ) AND recBuf[1] = 0 THEN
		icount0:=icount0+1;
	END_IF
	IF icount0 > 400 OR (GVL.Axis1Remote.iMode = 0 OR GVL.Axis1Remote.iMode = 0) THEN
		icount0 := 401;
		bEBN0Lock := FALSE;
	END_IF
END_IF

(* 旧版 0x7E 定界帧解析整段已注释 *)

                  
END_PROGRAM

FUNCTION_BLOCK Get_AZ
  VAR_INPUT
    uliRealTime : LREAL;  (* 当前时间戳，单位毫秒 *)
    lrStartTime : LREAL;  (* 任务起始时间，单位秒 *)
    rNodeTime1 : REAL;
    rNodeTime2 : REAL;
    rNodeTime3 : REAL;
    rNodeTime4 : REAL;
    rNodeTime5 : REAL;
    rEndTime : REAL;
    lrFun1 : ARRAY[0..10] OF LREAL;
    lrFun2 : ARRAY[0..10] OF LREAL;
    lrFun3 : ARRAY[0..10] OF LREAL;
    lrFun4 : ARRAY[0..10] OF LREAL;
    lrFun5 : ARRAY[0..10] OF LREAL;
    lrFun6 : ARRAY[0..10] OF LREAL;
  END_VAR
  VAR_OUTPUT
    lrFitResult : LREAL;
  END_VAR
  VAR
    rDelTime : REAL;
    rRealTime : LREAL;
  END_VAR

                    rRealTime := uliRealTime / 1000.0 - lrStartTime/1000.0;


IF rRealTime <= 0.0 THEN
	rDelTime := 0.0;
	lrFitResult := lrFun1[10];
ELSIF rRealTime <= rNodeTime1 THEN
    rDelTime := rRealTime - 0.0;
	lrFitResult := lrFun1[0] * EXPT(rDelTime,10) + lrFun1[1] * EXPT(rDelTime,9) + lrFun1[2] * EXPT(rDelTime,8) + lrFun1[3] * EXPT(rDelTime,7) + lrFun1[4] * EXPT(rDelTime,6) + lrFun1[5] * EXPT(rDelTime,5)
    + lrFun1[6] * EXPT(rDelTime,4) + lrFun1[7] * EXPT(rDelTime,3) + lrFun1[8] * EXPT(rDelTime,2) + lrFun1[9] * rDelTime + lrFun1[10];
ELSIF rRealTime <= rNodeTime2 THEN
    rDelTime := rRealTime - rNodeTime1;
    lrFitResult := lrFun2[0] * EXPT(rDelTime,10) + lrFun2[1] * EXPT(rDelTime,9) + lrFun2[2] * EXPT(rDelTime,8) + lrFun2[3] * EXPT(rDelTime,7) + lrFun2[4] * EXPT(rDelTime,6) + lrFun2[5] * EXPT(rDelTime,5)
    + lrFun2[6] * EXPT(rDelTime,4) + lrFun2[7] * EXPT(rDelTime,3) + lrFun2[8] * EXPT(rDelTime,2) + lrFun2[9] * rDelTime + lrFun2[10];
ELSIF rRealTime <= rNodeTime3 THEN
    rDelTime := rRealTime - rNodeTime2;
    lrFitResult := lrFun3[0] * EXPT(rDelTime,10) + lrFun3[1] * EXPT(rDelTime,9) + lrFun3[2] * EXPT(rDelTime,8) + lrFun3[3] * EXPT(rDelTime,7) + lrFun3[4] * EXPT(rDelTime,6) + lrFun3[5] * EXPT(rDelTime,5)
    + lrFun3[6] * EXPT(rDelTime,4) + lrFun3[7] * EXPT(rDelTime,3) + lrFun3[8] * EXPT(rDelTime,2) + lrFun3[9] * rDelTime + lrFun3[10];
ELSIF rRealTime <= rNodeTime4 THEN
    rDelTime := rRealTime - rNodeTime3;
    lrFitResult := lrFun4[0] * EXPT(rDelTime,10) + lrFun4[1] * EXPT(rDelTime,9) + lrFun4[2] * EXPT(rDelTime,8) + lrFun4[3] * EXPT(rDelTime,7) + lrFun4[4] * EXPT(rDelTime,6) + lrFun4[5] * EXPT(rDelTime,5)
    + lrFun4[6] * EXPT(rDelTime,4) + lrFun4[7] * EXPT(rDelTime,3) + lrFun4[8] * EXPT(rDelTime,2) + lrFun4[9] * rDelTime + lrFun4[10];
ELSIF rRealTime <= rNodeTime5 THEN
    rDelTime := rRealTime - rNodeTime4;
    lrFitResult := lrFun5[0] * EXPT(rDelTime,10) + lrFun5[1] * EXPT(rDelTime,9) + lrFun5[2] * EXPT(rDelTime,8) + lrFun5[3] * EXPT(rDelTime,7) + lrFun5[4] * EXPT(rDelTime,6) + lrFun5[5] * EXPT(rDelTime,5)
    + lrFun5[6] * EXPT(rDelTime,4) + lrFun5[7] * EXPT(rDelTime,3) + lrFun5[8] * EXPT(rDelTime,2) + lrFun5[9] * rDelTime + lrFun5[10];
ELSIF rRealTime <= rEndTime THEN
    rDelTime := rRealTime - rNodeTime5;
    lrFitResult := lrFun6[0] * EXPT(rDelTime,10) + lrFun6[1] * EXPT(rDelTime,9) + lrFun6[2] * EXPT(rDelTime,8) + lrFun6[3] * EXPT(rDelTime,7) + lrFun6[4] * EXPT(rDelTime,6) + lrFun6[5] * EXPT(rDelTime,5)
    + lrFun6[6] * EXPT(rDelTime,4) + lrFun6[7] * EXPT(rDelTime,3) + lrFun6[8] * EXPT(rDelTime,2) + lrFun6[9] * rDelTime + lrFun6[10];
ELSE
    rDelTime := rEndTime - rNodeTime5;
    lrFitResult := lrFun6[0] * EXPT(rDelTime,10) + lrFun6[1] * EXPT(rDelTime,9) + lrFun6[2] * EXPT(rDelTime,8) + lrFun6[3] * EXPT(rDelTime,7) + lrFun6[4] * EXPT(rDelTime,6) + lrFun6[5] * EXPT(rDelTime,5)
    + lrFun6[6] * EXPT(rDelTime,4) + lrFun6[7] * EXPT(rDelTime,3) + lrFun6[8] * EXPT(rDelTime,2) + lrFun6[9] * rDelTime + lrFun6[10];
END_IF

IF lrFitResult>270 THEN
	lrFitResult:=270;
ELSIF lrFitResult<-270 THEN
	lrFitResult:=-270;
END_IF
                  
END_FUNCTION_BLOCK

FUNCTION_BLOCK Get_AZ_1
  VAR_INPUT
    uliRealTime : LREAL;  (* 当前时间戳，单位毫秒 *)
    lrStartTime : LREAL;  (* 任务起始时间，单位秒 *)
    rNodeTime1 : REAL;
    rNodeTime2 : REAL;
    rNodeTime3 : REAL;
    rNodeTime4 : REAL;
    rNodeTime5 : REAL;
    rEndTime : REAL;
    lrFun1 : ARRAY[0..10] OF LREAL;
    lrFun2 : ARRAY[0..10] OF LREAL;
    lrFun3 : ARRAY[0..10] OF LREAL;
    lrFun4 : ARRAY[0..10] OF LREAL;
    lrFun5 : ARRAY[0..10] OF LREAL;
    lrFun6 : ARRAY[0..10] OF LREAL;
  END_VAR
  VAR_OUTPUT
    lrFitResult : LREAL;
  END_VAR
  VAR
    rDelTime : REAL;
    rRealTime : LREAL;
  END_VAR

                    rRealTime := uliRealTime / 1000.0 - lrStartTime/1000.0;


IF rRealTime <= 0.0 THEN
	rDelTime := 0.0;
	lrFitResult := lrFun1[10];
ELSIF rRealTime <= rNodeTime1 THEN
    rDelTime := rRealTime - 0.0;
	lrFitResult := lrFun1[0] * EXPT(rDelTime,10) + lrFun1[1] * EXPT(rDelTime,9) + lrFun1[2] * EXPT(rDelTime,8) + lrFun1[3] * EXPT(rDelTime,7) + lrFun1[4] * EXPT(rDelTime,6) + lrFun1[5] * EXPT(rDelTime,5)
    + lrFun1[6] * EXPT(rDelTime,4) + lrFun1[7] * EXPT(rDelTime,3) + lrFun1[8] * EXPT(rDelTime,2) + lrFun1[9] * rDelTime + lrFun1[10];
ELSIF rRealTime <= rNodeTime2 THEN
    rDelTime := rRealTime - rNodeTime1;
    lrFitResult := lrFun2[0] * EXPT(rDelTime,10) + lrFun2[1] * EXPT(rDelTime,9) + lrFun2[2] * EXPT(rDelTime,8) + lrFun2[3] * EXPT(rDelTime,7) + lrFun2[4] * EXPT(rDelTime,6) + lrFun2[5] * EXPT(rDelTime,5)
    + lrFun2[6] * EXPT(rDelTime,4) + lrFun2[7] * EXPT(rDelTime,3) + lrFun2[8] * EXPT(rDelTime,2) + lrFun2[9] * rDelTime + lrFun2[10];
ELSIF rRealTime <= rNodeTime3 THEN
    rDelTime := rRealTime - rNodeTime2;
    lrFitResult := lrFun3[0] * EXPT(rDelTime,10) + lrFun3[1] * EXPT(rDelTime,9) + lrFun3[2] * EXPT(rDelTime,8) + lrFun3[3] * EXPT(rDelTime,7) + lrFun3[4] * EXPT(rDelTime,6) + lrFun3[5] * EXPT(rDelTime,5)
    + lrFun3[6] * EXPT(rDelTime,4) + lrFun3[7] * EXPT(rDelTime,3) + lrFun3[8] * EXPT(rDelTime,2) + lrFun3[9] * rDelTime + lrFun3[10];
ELSIF rRealTime <= rNodeTime4 THEN
    rDelTime := rRealTime - rNodeTime3;
    lrFitResult := lrFun4[0] * EXPT(rDelTime,10) + lrFun4[1] * EXPT(rDelTime,9) + lrFun4[2] * EXPT(rDelTime,8) + lrFun4[3] * EXPT(rDelTime,7) + lrFun4[4] * EXPT(rDelTime,6) + lrFun4[5] * EXPT(rDelTime,5)
    + lrFun4[6] * EXPT(rDelTime,4) + lrFun4[7] * EXPT(rDelTime,3) + lrFun4[8] * EXPT(rDelTime,2) + lrFun4[9] * rDelTime + lrFun4[10];
ELSIF rRealTime <= rNodeTime5 THEN
    rDelTime := rRealTime - rNodeTime4;
    lrFitResult := lrFun5[0] * EXPT(rDelTime,10) + lrFun5[1] * EXPT(rDelTime,9) + lrFun5[2] * EXPT(rDelTime,8) + lrFun5[3] * EXPT(rDelTime,7) + lrFun5[4] * EXPT(rDelTime,6) + lrFun5[5] * EXPT(rDelTime,5)
    + lrFun5[6] * EXPT(rDelTime,4) + lrFun5[7] * EXPT(rDelTime,3) + lrFun5[8] * EXPT(rDelTime,2) + lrFun5[9] * rDelTime + lrFun5[10];
ELSIF rRealTime <= rEndTime THEN
    rDelTime := rRealTime - rNodeTime5;
    lrFitResult := lrFun6[0] * EXPT(rDelTime,10) + lrFun6[1] * EXPT(rDelTime,9) + lrFun6[2] * EXPT(rDelTime,8) + lrFun6[3] * EXPT(rDelTime,7) + lrFun6[4] * EXPT(rDelTime,6) + lrFun6[5] * EXPT(rDelTime,5)
    + lrFun6[6] * EXPT(rDelTime,4) + lrFun6[7] * EXPT(rDelTime,3) + lrFun6[8] * EXPT(rDelTime,2) + lrFun6[9] * rDelTime + lrFun6[10];
ELSE
    rDelTime := rEndTime - rNodeTime5;
    lrFitResult := lrFun6[0] * EXPT(rDelTime,10) + lrFun6[1] * EXPT(rDelTime,9) + lrFun6[2] * EXPT(rDelTime,8) + lrFun6[3] * EXPT(rDelTime,7) + lrFun6[4] * EXPT(rDelTime,6) + lrFun6[5] * EXPT(rDelTime,5)
    + lrFun6[6] * EXPT(rDelTime,4) + lrFun6[7] * EXPT(rDelTime,3) + lrFun6[8] * EXPT(rDelTime,2) + lrFun6[9] * rDelTime + lrFun6[10];
END_IF

IF lrFitResult>90 THEN
	lrFitResult:=90;
ELSIF lrFitResult<3 THEN
	lrFitResult:=3;
END_IF
                  
END_FUNCTION_BLOCK

FUNCTION_BLOCK AGCMaxSearch_PB_1
  VAR_INPUT
    bstart : BOOL;  (* 模块开始标识 *)
    rAGCNow : REAL;  (* 当前AGC值 *)
    btrig : BOOL;  (* 触发一次 *)
    rStepBiasNow : REAL;  (* 当前拉偏量 //用来判断此次搜索是否有效 *)
    bAutoTracking : BOOL;  (* 自跟踪标识 *)
    bStop : BOOL;  (* 满足ua ue很小 *)
    rCurrentPos : REAL;  (* 当前位置 *)
    rInterPos : REAL;  (* 插值位置 *)
  END_VAR
  VAR_OUTPUT
    rAGCMaxBias : REAL;  (* 输出AGC最强时的拉偏量 单位为° *)
    bSucess : BOOL;  (* 数出模块是否成功 *)
    rStepBias : REAL;  (* 步进量 *)
  END_VAR
  VAR
    ton : Standard.TON;
    rTrg : Standard.R_TRIG;  (* 初始化上升沿检测器 *)
    rAGCInit : REAL := 0;  (* 初始化AGC *)
    rPrevAGC : REAL := 0;  (* 上一步的AGC值 单位为V *)
    rBiasInit : REAL;  (* 初始化拉偏量 *)
    iCountStep : INT := 0;  (* 计步数 *)
    toN1 : Standard.Ton;  (* 计时器 定时触发上升沿 *)
    rDirection : INT := 1;
    rSearchNextStepTarget : REAL;  (* 搜索当前目标位置 单位为° *)
    rStep : REAL := 0.0003;  (* 步进值 *)
    rSensitivity : REAL := 0.05;  (* 反向灵敏度 *)
    iCountStopMax : INT := 20;  (* 停止计数上限 *)
    rLastDirection : INT;  (* 上一次方向，判断是否换向 *)
    iCountDirChange : INT;  (* 换向标识 *)
    rAGCMaxPos : REAL;  (* 信号最强位置 *)
    rAGCLastrecord : REAL;
    iStatus : INT;
    iCountStop1 : INT;  (* 第一阶段停止标识 (正向) *)
    iCountStop2 : INT;  (* (反向) *)
    rAGCMaxValue : REAL;  (* AGC最大值 *)
    iCountSearchRight : INT;  (* 搜索方向正确，提前结束标识 *)
    bSearchRight : BOOL;  (* 搜索正确标识 *)
    iCountBlockEnd : INT;  (* 用来计数确认已达到最强位置 *)
    iCountBlockEndMax : INT := 500;  (* 到位计数上限 *)
  END_VAR

                    
(*==============================================================================
  FB: AGCMaxSearch_PB_1（AGC 峰值搜索：单轴拉偏搜索）
  调用者: `Az_ctrl_1` / `El_ctrl_1`
  目标: 在指向(mode2)或程引(mode4)时，沿单轴正/负方向试探移动 rStepBias，
        找到使 AGC 最大的位置偏置 rAGCMaxBias，并在到位稳定后置 bSucess

  关键变量含义:
    rStepBias      — 当前偏置输出（逐步累加 rDirection*rStep）
    rAGCMaxBias    — 历史最大 AGC 对应的偏置
    rAGCInit       — 启动时 AGC 基线
    rSensitivity   — 判定“AGC 明显下降/上升”的阈值，用于决定停止/换向
    iCountDirChange— 换向次数；=2 后进入“回到峰值位置并等待稳定”阶段

  完成判定:
    - 偏置回到 rAGCMaxBias 后，(rInterPos+rStepBias) 与 rCurrentPos 误差持续小于 0.002
    - 持续计数超过 iCountBlockEndMax 后，再用 TON(1s) 确认稳定 → bSucess=TRUE
==============================================================================*)

rTrg(CLK:=bstart,Q=>);

IF rTrg.Q THEN
	rAGCInit:=rAGCNow;
	rAGCMaxValue:=rAGCNow;
	//rBiasInit:=rCurrentPos-rInterPos;//获取启动时的拉偏量
END_IF

IF bstart THEN
	//搜索换向两次
	IF iCountDirChange=2 THEN
		rSearchNextStepTarget:=rAGCMaxBias;
		IF rStepBias< rSearchNextStepTarget THEN 
			rStepBias:=rStepBias+rStep;
		ELSIF rStepBias> rSearchNextStepTarget THEN
			rStepBias:=rStepBias-rStep;
		ELSE
			rStepBias:=rStepBias;
		END_IF
		
		IF ABS((rInterPos+rStepBias)-rCurrentPos)<0.002 THEN //若位置达到最强位置，则输出成功 //可能只是路过这里,需要持续
			//需要判断稳定
			iCountBlockEnd:=iCountBlockEnd+1;
		ELSE
			iCountBlockEnd:=0;
		END_IF
		IF iCountBlockEnd>iCountBlockEndMax THEN
			iCountBlockEnd:=iCountBlockEndMax+1;
			//用TON1秒后触发
			ton(IN:=TRUE,PT:=T#1S,Q=>,ET=>);
		END_IF
		IF ton.Q THEN
			bSucess:=TRUE;
		END_IF
	ELSE
		rStepBias:=rStepBias+rDirection*rStep;
		IF rDirection<0 THEN
			//若是向小走
			IF rCurrentPos<rInterPos THEN
				IF rAGCNow<rAGCMaxValue-rSensitivity THEN
					iCountStop1:=iCountStop1+1;
					IF iCountStop1>iCountStopMax THEN
						iCountStop1:=iCountStopMax+1;
						IF bSearchRight THEN
							iCountDirChange:=2;
						ELSE
							iCountDirChange:=iCountDirChange+1;
						END_IF
						rDirection:=rDirection*(-1);
					END_IF
				ELSE
					iCountStop1:=0;	
				END_IF
				
				//新加的 测试第一阶段搜索正确后不进行第二次搜索
				IF rAGCNow>rAGCInit+rSensitivity THEN
					iCountSearchRight:=iCountSearchRight+1;
				ELSE
					iCountSearchRight:=0;
				END_IF
				IF iCountSearchRight>200 THEN
					iCountSearchRight:=201;
					bSearchRight:=TRUE;
				END_IF
				
			END_IF
		ELSE
			//若是向正走
			IF rCurrentPos>rInterPos THEN
				IF rAGCNow<rAGCMaxValue-rSensitivity THEN
					iCountStop2:=iCountStop2+1;
					IF iCountStop2>iCountStopMax THEN
						iCountStop2:=iCountStopMax+1;
						IF bSearchRight THEN
							iCountDirChange:=2;
						ELSE
							iCountDirChange:=iCountDirChange+1;
						END_IF
						rDirection:=rDirection*(-1);
					END_IF
				ELSE
					iCountStop2:=0;	
				END_IF
				
				//新加的
				IF rAGCNow>rAGCInit+rSensitivity THEN
					iCountSearchRight:=iCountSearchRight+1;
				ELSE
					iCountSearchRight:=0;
				END_IF
				IF iCountSearchRight>200 THEN
					iCountSearchRight:=201;
					bSearchRight:=TRUE;
				END_IF
				
			END_IF
		END_IF
		(*
		IF rAGCNow<rAGCInit-0.05 THEN
			iCountStop1:=iCountStop1+1;
			IF iCountStop1>150 THEN
				iCountDirChange:=iCountDirChange+1;
				rDirection:=rDirection*(-1);
			END_IF
		ELSE
			iCountStop1:=0;	
		END_IF
		*)
		
		 // 记录最强信号的拉偏量和值
		//IF rAGCNow >= rAGCInit AND rAGCNow> rAGCMaxValue THEN
		IF  rAGCNow> rAGCMaxValue THEN
			rAGCMaxBias := rStepBias;
			rAGCMaxValue := rAGCNow;
		END_IF
	END_IF
ELSE
	rStepBias:=0;
	//清空变量
	iCountDirChange:=0;
	rAGCInit:=0;
	rAGCMaxValue:=0;
	rAGCMaxBias:=0;
	rDirection:=1;
	iCountStop1:=0;
	iCountStop2:=0;
	ton(IN:=FALSE,PT:=T#1S,Q=>,ET=>);
	//rStepBias:=0;
	rSearchNextStepTarget:=0;
	bSucess:=FALSE;
	iCountSearchRight:=0;
	bSearchRight:=FALSE;
	iCountBlockEnd:=0;
END_IF


(*
IF rStepBias< rSearchNextStepTarget THEN 
	rStepBias:=rStepBias+rStep;
ELSIF rStepBias> rSearchNextStepTarget THEN
	rStepBias:=rStepBias-rStep;
ELSE
	rStepBias:=rStepBias;
END_IF*)
                  
END_FUNCTION_BLOCK

PROGRAM GPRMC_1
  VAR
    com_init : gcan.FB_Com_Init;  (* gcan.FB_Com_Init为串口初始化功能块，可设定串口端口号，串口波特率等参数 *)
    com_read : gcan.FB_Com_Read;  (* gcan.FB_Com_Read为串口接收功能块，用于通过接收串口发送给PLC的数据 *)
    com_write : gcan.FB_Com_Write;  (* gcan.FB_Com_Write为串口发送功能块，用于发送串口数据 *)
    m_uiError : UINT;  (* 用于承接功能块中报错引脚错误信息的变量 *)
    m_out : BOOL;  (* 用于承接功能块中完成标志引脚数据的变量 *)
    isFirst : BOOL := TRUE;  (* 用于判断初始化只执行一次的逻辑 *)
    mPort : BYTE;  (* 程序中用作设定串口端口号 *)
    recSize : UINT;  (* 接收数据长度，单位：字节 *)
    recBuf : ARRAY[0..101] OF BYTE;  (* 用于存放接收到的串口数据的数组 *)
    sum_i : INT;
    checksum : BYTE;
    iYear : INT;
    iMonth : INT;
    iDay : INT;
    iHour : INT;
    iMinute : INT;
    iSecond : INT;
    strDateTimeNow : STRING;
    gnssTimestamp : ULINT;
    gnssTimestamplast : ULINT;
    icount : INT;
    high4 : BYTE;
    low4 : BYTE;
  END_VAR
  VAR_INPUT
    EN_in_1 : BOOL;
  END_VAR

                    (*==============================================================================
  PRG: GPRMC_1（GNSS 串口接收与 NMEA 时间解析）
  任务: SerialCom 5ms
  硬件: GCAN 模块串口 mPort=1（232），115200 8N1
  作用:
    - 读 GNSS 模块输出的 NMEA 报文（GPRMC 等，帧头 ASCII '$'=36）
    - 从固定偏移解析 UTC 日期时间，+8 转为北京时间
    - 写入 GVL.stGNSS_Timestap（毫秒 ULINT），供 TimeAdd / RealTimePosCal 使用
  下游:
    TimeAdd.icount — 秒未变时累加，用于 GNSS 丢帧时的 10ms 插值
    RealTimePosCal — GVL.dRealTime := stGNSS_Timestap + 10*TimeAdd.icount
==============================================================================*)


////////////////////////////////////////////////////////////////////////////////////////
//串口接收GPRMC报文解析
//日期：2024/08/25
//版本：V1.1
/////////////////////////////////////////////////////////////////////////////////////////

mPort:=1;								//串口端口号设定，GCAN-PLC-400、GCAN-PLC-510、GCAN-PLC-511，1为232，2为485
										//GCAN-PLC-324、GCAN-PLC-326，1为第一路485，2为第2路485
IF isFirst THEN
	com_init(							//串口初始化功能块
	EN_IN:=TRUE,						//串口初始化功能块使能
	xEnable:=TRUE,						//串口功能使能
	bPort:=mPort,						//串口端口号设定
	uiBaudrate:=115200,					//串口波特率设定
	bParity:=0,							//串口奇偶校验设定，0为无校验，1为奇校验，2为偶检验
	bDatabits:=8,						//数据位设定
	bStopbits:=1,						//停止位设定
	EN_OUT=>m_out,						//串口初始化功能块执行完成标志位
	uiError=>m_uiError);				//串口初始化功能块执行错误信息
	isfirst:=FALSE;						//执行一次初始化后关闭IF的条件使其之后进入ELSE程序段运行

ELSE
	
		com_read(						//串口读取功能块
		EN_in:=TRUE,					//读取功能块使能，为TRUE执行读取
		bPort:=mPort,					//串口端口号设定
		p_brxdata:=ADR(recBuf),			//读取到的串口数据引脚为指针类型，使用ADR()指向自建数组将数据存放到数组中
		uiMaxsize:=204,					//设定最大读取长度
		EN_out=>m_out,					//串口读取功能块执行完成标志位******功能块执行完成不代表接收完成********
		uiRecSize=>recSize,				//串口接收数据长度，单位：字节，大于0时说明接收到数据可用于判断是否接收
		uierror=>m_uierror);			//串口读取功能块执行错误信息
										//从数组recBuf里取数据，解析出年、月、日、时、分、秒
		//有效判定(A)+和校验(hh),前 4bit和后 4bit的 16 进制数分别以 ASCII 码表示(0~9,A~F)，高位在前。
		IF 	recBuf[0] = 36 THEN
(*			checksum := 16#00;
			FOR sum_i:=1 TO 74 BY 1 DO
				checksum:= checksum XOR recBuf[sum_i];
			END_FOR
			high4 := (SHR(checksum, 4) AND 16#0F)+16#30;
			low4 := (checksum AND 16#0F)+16#30;
			IF recBuf[76]= high4 AND recBuf[77]= low4 THEN 
*)		

			iYear:=BYTE_TO_INT(recBuf[23]-48)*1000+BYTE_TO_INT(recBuf[24]-48)*100+BYTE_TO_INT(recBuf[25]-48)*10+BYTE_TO_INT(recBuf[26]-48);
			iMonth:=BYTE_TO_INT(recBuf[20]-48)*10+BYTE_TO_INT(recBuf[21]-48);
			iDay:=BYTE_TO_INT(recBuf[17]-48)*10+BYTE_TO_INT(recBuf[18]-48);
			iHour:=BYTE_TO_INT(recBuf[7]-48)*10+BYTE_TO_INT(recBuf[8]-48)+8;
			iMinute:=BYTE_TO_INT(recBuf[9]-48)*10+BYTE_TO_INT(recBuf[10]-48);
			iSecond:=BYTE_TO_INT(recBuf[11]-48)*10+BYTE_TO_INT(recBuf[12]-48);
			
			// 计算时间戳		
			
			strDateTimeNow := CONCAT(STR1 := 'DT#', STR2 := INT_TO_STRING(iYear));
			strDateTimeNow := CONCAT(STR1 := strDateTimeNow, STR2 := '-');
			strDateTimeNow := CONCAT(STR1 := strDateTimeNow, STR2 := INT_TO_STRING(iMonth));
			strDateTimeNow := CONCAT(STR1 := strDateTimeNow, STR2 := '-');
			strDateTimeNow := CONCAT(STR1 := strDateTimeNow, STR2 := INT_TO_STRING(iDay));
			strDateTimeNow := CONCAT(STR1 := strDateTimeNow, STR2 := '-');
			strDateTimeNow := CONCAT(STR1 := strDateTimeNow, STR2 := INT_TO_STRING(iHour));
			strDateTimeNow := CONCAT(STR1 := strDateTimeNow, STR2 := ':');
			strDateTimeNow := CONCAT(STR1 := strDateTimeNow, STR2 := INT_TO_STRING(iMinute));
			strDateTimeNow := CONCAT(STR1 := strDateTimeNow, STR2 := ':');
			strDateTimeNow := CONCAT(STR1 := strDateTimeNow, STR2 := INT_TO_STRING(iSecond));
			(*
			gnssTimestamplast:=gnssTimestamp;
			
			
			*)
			gnssTimestamp := DT_TO_ULINT(TO_DT(strDateTimeNow)) * 1000;
			GVL.stGNSS_Timestap := gnssTimestamp;
		END_IF
		(*
		IF gnssTimestamplast<>gnssTimestamp THEN
			icount:=0;
		ELSE
			icount:=icount+1;
		END_IF
		*)
		


(*	IF recsize>0 THEN					//如果接收到串口数据
		
		com_write(						//串口发送功能块
		EN_IN:=TRUE,					//串口发送功能块使能，发送机制：当使能为TRUE时，PLC程序每周期运行到此处就执行一次发送
		bPort:=mPort,					//串口端口号设定
		p_bTxdata:=ADR(recbuf),			//将接收存放到数组中的数据发送出去******若发送其它数据，自建另一数组用于存放发送数据即可
		uiTxsize:=recsize,				//发送长度为接收到的数据长度******若发送其它长度，自行填写所需长度即可
		EN_OUT=>m_out,					//串口发送功能块执行完成标志位
		uierror=>m_uierror);			//串口发送功能块执行错误信息
			
	END_IF
*)	
END_IF
                  
END_PROGRAM

PROGRAM GetACUTime
  VAR
    tp : TP;  (* 脉冲定时器 *)
    toggle : BOOL := FALSE;  (* 当前输出状态 *)
    clk : BOOL := FALSE;  (* 方波输出 *)
    tick_ms : TIME := TIME#500ms;  (* 高电平/低电平持续时间 *)
    Result : RTS_IEC_RESULT;
    stUTC_Timestamp : SYSTIME;
    dRTime : ULINT;  (* 上位机外部时间 单位ns Unix时间戳，起点是1970-1-1 0:0:0 *)
    dModbusTime : ULINT;  (* Modbus临时外部时间 *)
    iCountRemote : INT;  (* 上位机锁定判断时间常数 *)
    dCountRemote : ULINT;  (* 上位机时间滑动平均常数 *)
    dLastRTime : ULINT;  (* 上位机上一次外部时间 单位ns Unix时间戳，起点是1970-1-1 0:0:0 *)
    iDiffRTime : DINT;  (* 上位机时间差值 *)
    dDelRTime : LINT;
    dMeanDelRTime : LINT;
    rTriger : Standard.R_TRIG;  (* 上升沿触发器 *)
    iDiff : DINT;  (* 实际时间差值 *)
    iDiffLocal : DINT;  (* 本地时间差值 *)
    iDiffETime : DINT;  (* 外部时间差值 *)
    ulACUTimeStamp : ULINT;
  END_VAR

                    
// 每次TP结束时翻转状态
IF NOT tp.Q THEN
    toggle := NOT toggle;
    tp.IN := TRUE;
    tp.PT := tick_ms;
ELSE
    tp.IN := FALSE;
END_IF

tp();

Result := SysTimeRtcHighResGet(stUTC_Timestamp);
rTriger(CLK:=toggle);
IF rTriger.Q THEN
	dRTime := modbus_slave.UTC_New;
	iDiffRTime:=ULINT_TO_DINT(dRTime-dLastRTime);
	IF ABS(iDiffRTime)>500 THEN //两次PTP时间差如果大于500毫秒,则判断为上位机时间失锁
		iCountRemote:=0;
		dCountRemote:=0;
		GVL.bRemoteTimeLock:=FALSE;
	ELSE//否则判断为上位机时间锁定并累计1分钟
		iCountRemote:=iCountRemote+1;
	END_IF
	
	IF iCountRemote>=20 THEN //累计20s认为时间可用
		iCountRemote:=20;
		dDelRTime := TO_ULINT(stUTC_Timestamp) - (dRTime + 8 * 3600 *1000);
		GVL.bRemoteTimeLock:=TRUE;
		//对外部和本机时间差做1分钟的均值滤波
	END_IF
	//GVL.dRemoteTime:=stUTC_Timestamp*1000000 - dMeanDelRTime;
	dLastRTime:=dRTime;
	(*
	IF GVL.bRemoteTimeLock THEN
		dCountRemote:= dCountRemote + 1;
		IF dCountRemote < 10000 THEN
			dMeanDelRTime := (dMeanDelRTime*(dCountRemote-1) + dDelRTime)/dCountRemote;
		ELSE
			dCountRemote := 10000;
			dMeanDelRTime := (dMeanDelRTime*(dCountRemote-1) + dDelRTime)/dCountRemote; 	
			//iDiff:=ULINT_TO_DINT(Gvl.dPTPCSTTime-dLastCSTtime);
			//dLastCSTtime:=dCSTTime;
		END_IF
	END_IF
	*)
END_IF

ulACUTimeStamp := stUTC_Timestamp - dDelRTime;
                  
END_PROGRAM

PROGRAM XPTOD_SerialCom
  VAR
    com_init : gcan.FB_Com_Init;  (* gcan.FB_Com_Init为串口初始化功能块，可设定串口端口号，串口波特率等参数 *)
    com_read : gcan.FB_Com_Read;  (* gcan.FB_Com_Read为串口接收功能块，用于通过接收串口发送给PLC的数据 *)
    com_write : gcan.FB_Com_Write;  (* gcan.FB_Com_Write为串口发送功能块，用于发送串口数据 *)
    m_uiError : UINT;  (* 用于承接功能块中报错引脚错误信息的变量 *)
    m_out : BOOL;  (* 用于承接功能块中完成标志引脚数据的变量 *)
    isFirst : BOOL := TRUE;  (* 用于判断初始化只执行一次的逻辑 *)
    mPort : BYTE;  (* 程序中用作设定串口端口号 *)
    recSize : UINT;  (* 接收数据长度，单位：字节 *)
    recBuf : ARRAY[0..239] OF BYTE;  (* 用于存放接收到的串口数据的数组 *)
    iYear : INT;  (* 年 *)
    iMonth : INT;  (* 月 *)
    iDay : INT;  (* 日 *)
    iHour : INT;  (* 时 *)
    iMinute : INT;  (* 分 *)
    iSecond : INT;  (* 秒 *)
    bChecksumValid : BOOL := FALSE;  (* 校验和 *)
    nFrameHeadPos : INT := 0;  (* 帧头索引 *)
    nPos : INT;  (* 帧头位置 *)
    nChecksumRx : BYTE := 0;  (* 和校验 *)
    strDateTimeNow : STRING;
    gnssTimestamp : ULINT;
    gnssTimestamplast : ULINT;
    icount : INT;
  END_VAR

                    ////////////////////////////////////////////////////////////////////////////////////////
//串口接收TOD报文解析
//日期：2025/05/15
//版本：V1.1
/////////////////////////////////////////////////////////////////////////////////////////

mPort:=1;                                                                //串口端口号设定，GCAN-PLC-400、GCAN-PLC-510、GCAN-PLC-511，1为232，2为485
                                                                                //GCAN-PLC-324、GCAN-PLC-326，1为第一路485，2为第2路485
IF isFirst THEN
        com_init(                                                        //串口初始化功能块
        EN_IN:=TRUE,                                                //串口初始化功能块使能
        xEnable:=TRUE,                                                //串口功能使能
        bPort:=mPort,                                                //串口端口号设定
        uiBaudrate:=115200,                                        //串口波特率设定
        bParity:=0,                                                        //串口奇偶校验设定，0为无校验，1为奇校验，2为偶检验
        bDatabits:=8,                                                //数据位设定
        bStopbits:=1,                                                //停止位设定
        EN_OUT=>m_out,                                                //串口初始化功能块执行完成标志位
        uiError=>m_uiError);                                //串口初始化功能块执行错误信息
        isfirst:=FALSE;                                                //执行一次初始化后关闭IF的条件使其之后进入ELSE程序段运行

ELSE
        
                com_read(                                                //串口读取功能块
                EN_in:=TRUE,                                        //读取功能块使能，为TRUE执行读取
                bPort:=mPort,                                        //串口端口号设定
                p_brxdata:=ADR(recBuf),                        //读取到的串口数据引脚为指针类型，使用ADR()指向自建数组将数据存放到数组中
                uiMaxsize:=240,                                        //设定最大读取长度
                EN_out=>m_out,                                        //串口读取功能块执行完成标志位******功能块执行完成不代表接收完成********
                uiRecSize=>recSize,                                //串口接收数据长度，单位：字节，大于0时说明接收到数据可用于判断是否接收
                uierror=>m_uierror);                        //串口读取功能块执行错误信息
                // 查找帧头 $X (36, 88)
                FOR nPos := 1 TO 240 DO
                        IF recBuf[nPos] = 36 AND recBuf[nPos + 1] = 88 THEN
                                nFrameHeadPos := nPos;
                                EXIT;
                        END_IF
                END_FOR
                //解析时间日期 
                IF nFrameHeadPos + 26 <= 240 THEN
                        iYear:=BYTE_TO_INT(recBuf[nFrameHeadPos+23]-48)*1000+BYTE_TO_INT(recBuf[nFrameHeadPos+24]-48)*100+BYTE_TO_INT(recBuf[nFrameHeadPos+25]-48)*10+BYTE_TO_INT(recBuf[26]-48);
                        iMonth:=BYTE_TO_INT(recBuf[nFrameHeadPos+20]-48)*10+BYTE_TO_INT(recBuf[nFrameHeadPos+21]-48);
                        iDay:=BYTE_TO_INT(recBuf[nFrameHeadPos+17]-48)*10+BYTE_TO_INT(recBuf[nFrameHeadPos+18]-48);
                        iHour:=BYTE_TO_INT(recBuf[nFrameHeadPos+7]-48)*10+BYTE_TO_INT(recBuf[nFrameHeadPos+8]-48)+8;
                        iMinute:=BYTE_TO_INT(recBuf[nFrameHeadPos+9]-48)*10+BYTE_TO_INT(recBuf[nFrameHeadPos+10]-48);
                        iSecond:=BYTE_TO_INT(recBuf[nFrameHeadPos+11]-48)*10+BYTE_TO_INT(recBuf[nFrameHeadPos+12]-48);
                        // 计算时间戳                
                        
                        strDateTimeNow := CONCAT(STR1 := 'DT#', STR2 := INT_TO_STRING(iYear));
                        strDateTimeNow := CONCAT(STR1 := strDateTimeNow, STR2 := '-');
                        strDateTimeNow := CONCAT(STR1 := strDateTimeNow, STR2 := INT_TO_STRING(iMonth));
                        strDateTimeNow := CONCAT(STR1 := strDateTimeNow, STR2 := '-');
                        strDateTimeNow := CONCAT(STR1 := strDateTimeNow, STR2 := INT_TO_STRING(iDay));
                        strDateTimeNow := CONCAT(STR1 := strDateTimeNow, STR2 := '-');
                        strDateTimeNow := CONCAT(STR1 := strDateTimeNow, STR2 := INT_TO_STRING(iHour));
                        strDateTimeNow := CONCAT(STR1 := strDateTimeNow, STR2 := ':');
                        strDateTimeNow := CONCAT(STR1 := strDateTimeNow, STR2 := INT_TO_STRING(iMinute));
                        strDateTimeNow := CONCAT(STR1 := strDateTimeNow, STR2 := ':');
                        strDateTimeNow := CONCAT(STR1 := strDateTimeNow, STR2 := INT_TO_STRING(iSecond));
                        
                        gnssTimestamplast:=gnssTimestamp;
                        gnssTimestamp := DT_TO_ULINT(TO_DT(strDateTimeNow)) * 1000;
                        GVL.stGNSS_Timestap := gnssTimestamp;                        
                END_IF
                
                IF gnssTimestamplast<>gnssTimestamp THEN
                        icount:=0;
                ELSE
                        icount:=icount+1;
                END_IF        
END_IF
                  
END_PROGRAM

PROGRAM GPRMC_1_1
  VAR
    com_init : gcan.FB_Com_Init;  (* gcan.FB_Com_Init为串口初始化功能块，可设定串口端口号，串口波特率等参数 *)
    com_read : gcan.FB_Com_Read;  (* gcan.FB_Com_Read为串口接收功能块，用于通过接收串口发送给PLC的数据 *)
    com_write : gcan.FB_Com_Write;  (* gcan.FB_Com_Write为串口发送功能块，用于发送串口数据 *)
    m_uiError : UINT;  (* 用于承接功能块中报错引脚错误信息的变量 *)
    m_out : BOOL;  (* 用于承接功能块中完成标志引脚数据的变量 *)
    isFirst : BOOL := TRUE;  (* 用于判断初始化只执行一次的逻辑 *)
    mPort : BYTE;  (* 程序中用作设定串口端口号 *)
    recSize : UINT;  (* 接收数据长度，单位：字节 *)
    recBuf : ARRAY[0..120] OF BYTE;  (* 用于存放接收到的串口数据的数组 *)
    iYear : INT;  (* 年 *)
    iMonth : INT;  (* 月 *)
    iDay : INT;  (* 日 *)
    iHour : INT;  (* 时 *)
    iMinute : INT;  (* 分 *)
    iSecond : INT;  (* 秒 *)
    bChecksumValid : BOOL := FALSE;  (* 校验和 *)
    nFrameHeadPos : INT := 0;  (* 帧头索引 *)
    nPos : INT;  (* 帧头位置 *)
    nChecksumRx : BYTE := 0;  (* 和校验 *)
    strDateTimeNow : STRING;
    gnssTimestamp : ULINT;
    gnssTimestamplast : ULINT;
    icount : INT;
  END_VAR

                    ////////////////////////////////////////////////////////////////////////////////////////
//串口接收TOD报文解析
//日期：2025/05/15
//版本：V1.1
/////////////////////////////////////////////////////////////////////////////////////////

mPort:=1;                                                                //串口端口号设定，GCAN-PLC-400、GCAN-PLC-510、GCAN-PLC-511，1为232，2为485
                                                                                //GCAN-PLC-324、GCAN-PLC-326，1为第一路485，2为第2路485
IF isFirst THEN
        com_init(                                                        //串口初始化功能块
        EN_IN:=TRUE,                                                //串口初始化功能块使能
        xEnable:=TRUE,                                                //串口功能使能
        bPort:=mPort,                                                //串口端口号设定
        uiBaudrate:=115200,                                        //串口波特率设定
        bParity:=0,                                                        //串口奇偶校验设定，0为无校验，1为奇校验，2为偶检验
        bDatabits:=8,                                                //数据位设定
        bStopbits:=1,                                                //停止位设定
        EN_OUT=>m_out,                                                //串口初始化功能块执行完成标志位
        uiError=>m_uiError);                                //串口初始化功能块执行错误信息
        isfirst:=FALSE;                                                //执行一次初始化后关闭IF的条件使其之后进入ELSE程序段运行

ELSE
        
                com_read(                                                //串口读取功能块
                EN_in:=TRUE,                                        //读取功能块使能，为TRUE执行读取
                bPort:=mPort,                                        //串口端口号设定
                p_brxdata:=ADR(recBuf),                        //读取到的串口数据引脚为指针类型，使用ADR()指向自建数组将数据存放到数组中
                uiMaxsize:=240,                                        //设定最大读取长度
                EN_out=>m_out,                                        //串口读取功能块执行完成标志位******功能块执行完成不代表接收完成********
                uiRecSize=>recSize,                                //串口接收数据长度，单位：字节，大于0时说明接收到数据可用于判断是否接收
                uierror=>m_uierror);                        //串口读取功能块执行错误信息
                // 查找帧头 $X (36, 88)
                FOR nPos := 0 TO 119 DO
                        IF recBuf[nPos] = 36 AND recBuf[nPos + 1] = 88 THEN
                                nFrameHeadPos := nPos;
                                EXIT;
                        END_IF
                END_FOR
                //解析时间日期 
                IF nFrameHeadPos + 26 <= 120 THEN
                        iYear:=BYTE_TO_INT(recBuf[nFrameHeadPos+23]-48)*1000+BYTE_TO_INT(recBuf[nFrameHeadPos+24]-48)*100+BYTE_TO_INT(recBuf[nFrameHeadPos+25]-48)*10+BYTE_TO_INT(recBuf[26]-48);
                        iMonth:=BYTE_TO_INT(recBuf[nFrameHeadPos+20]-48)*10+BYTE_TO_INT(recBuf[nFrameHeadPos+21]-48);
                        iDay:=BYTE_TO_INT(recBuf[nFrameHeadPos+17]-48)*10+BYTE_TO_INT(recBuf[nFrameHeadPos+18]-48);
                        iHour:=BYTE_TO_INT(recBuf[nFrameHeadPos+7]-48)*10+BYTE_TO_INT(recBuf[nFrameHeadPos+8]-48)+8;
                        iMinute:=BYTE_TO_INT(recBuf[nFrameHeadPos+9]-48)*10+BYTE_TO_INT(recBuf[nFrameHeadPos+10]-48);
                        iSecond:=BYTE_TO_INT(recBuf[nFrameHeadPos+11]-48)*10+BYTE_TO_INT(recBuf[nFrameHeadPos+12]-48);
                        // 计算时间戳                
                        
                        strDateTimeNow := CONCAT(STR1 := 'DT#', STR2 := INT_TO_STRING(iYear));
                        strDateTimeNow := CONCAT(STR1 := strDateTimeNow, STR2 := '-');
                        strDateTimeNow := CONCAT(STR1 := strDateTimeNow, STR2 := INT_TO_STRING(iMonth));
                        strDateTimeNow := CONCAT(STR1 := strDateTimeNow, STR2 := '-');
                        strDateTimeNow := CONCAT(STR1 := strDateTimeNow, STR2 := INT_TO_STRING(iDay));
                        strDateTimeNow := CONCAT(STR1 := strDateTimeNow, STR2 := '-');
                        strDateTimeNow := CONCAT(STR1 := strDateTimeNow, STR2 := INT_TO_STRING(iHour));
                        strDateTimeNow := CONCAT(STR1 := strDateTimeNow, STR2 := ':');
                        strDateTimeNow := CONCAT(STR1 := strDateTimeNow, STR2 := INT_TO_STRING(iMinute));
                        strDateTimeNow := CONCAT(STR1 := strDateTimeNow, STR2 := ':');
                        strDateTimeNow := CONCAT(STR1 := strDateTimeNow, STR2 := INT_TO_STRING(iSecond));
                        
                        gnssTimestamplast:=gnssTimestamp;
                        gnssTimestamp := DT_TO_ULINT(TO_DT(strDateTimeNow)) * 1000;
                        GVL.stGNSS_Timestap := gnssTimestamp;                        
                END_IF
                
                IF gnssTimestamplast<>gnssTimestamp THEN
                        icount:=0;
                ELSE
                        icount:=icount+1;
                END_IF        
END_IF
                  
END_PROGRAM

FUNCTION_BLOCK SpiralScan
  VAR_INPUT
    enable : BOOL;  (* 启动使能 *)
    delta : REAL;  (* 扫描范围（°） *)
    delta1 : REAL;
    n_steps : REAL;  (* 每周期步长（°） *)
    agc : REAL;  (* 当前AGC *)
    locked : BOOL;  (* 锁定状态 *)
    AzError : REAL;
    ELError : REAL;
    bTrackState : BOOL;
  END_VAR
  VAR_OUTPUT
    azimuth : REAL;  (* 当前方位角输出 *)
    elevation : REAL;  (* 当前俯仰角输出 *)
    done : BOOL;  (* 扫描完成标志 *)
    bType : BOOL;  (* 是否提前结束，1是，0否 *)
  END_VAR
  VAR
    lock_count : INT := 0;
    best_agc : REAL := 0.0;
    best_az : REAL := 0.0;
    best_el : REAL := 0.0;
    bInit : BOOL;
    icount0 : INT := 0;
    icount1 : INT := 0;
    x : REAL := 0.0;
    y : REAL := 0.0;
    dx : REAL := 1.0;
    dy : REAL := 0.0;
    step_len : REAL := 1.0;
    step_count : REAL := 0.0;
    segment_progress : REAL := 0.0;
    move_count : REAL := 1.0;
    state : INT := 0;
    az0 : REAL := 0.0;
    el0 : REAL := 0.0;
    az1 : REAL := 0.0;
    el1 : REAL := 0.0;
    segment_az_step : REAL := 0.0;
    segment_el_step : REAL := 0.0;
    side_repeat : REAL := 0.0;
    icountInit : INT := 0;
    iSearchMax : INT;
    iCountSearch : INT;
    rTemp : REAL;
  END_VAR

                    

(*==============================================================================
  FB: SpiralScan（捕获扫描：矩形/十字格点扫描）
  调用者: `SecurityCheck`（段 11），当双轴程引 mode4 且未自跟踪时，用于“捕获目标”

  输入:
    enable      — 扫描使能（由 SecurityCheck 组合条件给出）
    delta       — 方位扫描半幅（deg）
    delta1      — 俯仰扫描半幅（deg），通过 rTemp=delta1/delta 与方位步进联动
    n_steps     — 单步步长（deg）
    agc         — 当前 AGC（越大越好）
    locked      — 锁定判定（Chan1EB_N0/误差电压门限等）
    AzError/ElError — 当前误差（用于记录 best_az/best_el，输出为 -Error）
    bTrackState — 已经进入自跟踪时为 TRUE，则直接 done

  	输出:
    azimuth/elevation — 给 `SecurityCheck.az_out/el_out` 的修正量
    done             — 扫描结束（提前锁定或扫描完毕）
    bType            — TRUE: 提前结束/锁定路径；FALSE: 扫描完毕输出最佳格点

  	状态机:
    state=0 等待锁定采样（避免瞬时锁定误触发）
    state=1 扫描：按 4 个象限依次走格点（iCountSearch 1..4*iSearchMax）
    state=2 提前锁定完成（保持 best_* 或 -Error）
    state=3 扫描完毕（输出 best_*）
==============================================================================*)




IF NOT enable THEN
    state := 0;
    azimuth := 0.0;
    elevation := 0.0;
    done := FALSE;
	lock_count := 0;
	icount0 := 0;
	segment_progress := 0.0;
	bInit := FALSE;
	best_agc := 0.0;
    best_az := 0.0;
    best_el := 0.0;
	icountInit := 0;
	iCountSearch := 0;
	
ELSE
    CASE state OF
        // --- 状态0：判断是否已锁定 ---
        0:
			IF NOT bTrackState THEN
				icountInit := icountInit + 1;
				IF icountInit >= 100 THEN
					icountInit := 101;
					icount0 := icount0 + 1;
					IF locked THEN
						lock_count := lock_count + 1;
					END_IF;
					IF icount0 >= 100 THEN
						IF lock_count >= 10 THEN
							done := TRUE;
							state := 2;   // 提前结束
							lock_count := 0;
						ELSE
							state := 1;   // 转入扫描
							lock_count := 0;
						END_IF;
					END_IF
				END_IF
			ELSE
				done := TRUE;
				state := 2;   // 提前结束
				lock_count := 0;
			END_IF
        1:
            IF NOT bTrackState THEN
				IF NOT bInit THEN
					x := 0.0; y := 0.0;
					dx := 1.0; dy := 0.0;
					step_len := 1.0;
					step_count := 0.0;
					move_count := 1.0;
					side_repeat := 0.0;
					az0 := 0.0; el0 := 0.0;
					az1 := delta * x;
					el1 := delta * y;
					segment_progress := 0.0;
					bInit := TRUE;
					iSearchMax := TO_INT(delta / n_steps);
					IF ABS(delta) < 1E-5 THEN
						rTemp := 0;
					ELSE
						rTemp := delta1 / delta;
					END_IF
				ELSE
					iCountSearch := iCountSearch + 1;
					IF iCountSearch <= iSearchMax THEN
						azimuth := n_steps * iCountSearch;
						elevation := n_steps * iCountSearch * rTemp;
					ELSIF iCountSearch <= 2 * iSearchMax THEN
						azimuth := delta - n_steps * (iCountSearch - iSearchMax);
						elevation := (delta - n_steps * (iCountSearch - iSearchMax)) * rTemp;
					ELSIF iCountSearch <= 3 * iSearchMax THEN
						azimuth := -1*n_steps * (iCountSearch - 2*iSearchMax);
						elevation := (-1*n_steps * (iCountSearch - 2*iSearchMax)) * rTemp;
					ELSIF iCountSearch < 4 * iSearchMax THEN
						azimuth := n_steps * (iCountSearch - 3*iSearchMax) - delta;
						elevation := (n_steps * (iCountSearch - 3*iSearchMax) - delta) * rTemp;
					END_IF
					
					
					IF agc > best_agc THEN
						best_agc := agc;
						best_az := -Azerror;
						best_el := -elError;
					END_IF;
					
					IF iCountSearch >= 4 * iSearchMax THEN
						state := 3;
					ELSE
						IF locked THEN
						   lock_count := lock_count + 1;
						ELSE
						   lock_count := 0;
						END_IF
						IF lock_count >= 10 THEN
						   done := TRUE;
						   state := 2;   // 提前结束
						   azimuth := best_az;
						   elevation := best_el;
						END_IF
					END_IF
				END_IF
			ELSE
				done := TRUE;
				state := 2;   // 提前结束
				azimuth := -Azerror;
				elevation := -elError;
			END_IF
        // --- 状态2：提前锁定完成 ---
        2:
            // 保持当前位置即可
            done := TRUE;
			

        // --- 状态3：完成，输出最佳格点 ---
        3:
            azimuth := best_az;
            elevation := best_el;
            done := TRUE;

    END_CASE
	
	IF state = 3 THEN
		bType := FALSE;
	ELSE
		bType := TRUE;
	END_IF
	
	IF ABS(delta1) < 1E-4 THEN
		elevation := 0; 
	END_IF
END_IF;
                  
END_FUNCTION_BLOCK

FUNCTION_BLOCK SpiralScan_1
  VAR_INPUT
    enable : BOOL;  (* 启动使能 *)
    delta : REAL;  (* 每格步长（°） *)
    n_steps : REAL;  (* 每格分段周期数 *)
    agc : REAL;  (* 当前AGC *)
    locked : BOOL;  (* 锁定状态 *)
    AzError : REAL;
    ELError : REAL;
  END_VAR
  VAR_OUTPUT
    azimuth : REAL;  (* 当前方位角输出 *)
    elevation : REAL;  (* 当前俯仰角输出 *)
    done : BOOL;  (* 扫描完成标志 *)
    bType : BOOL;  (* 是否提前结束，1是，0否 *)
  END_VAR
  VAR
    lock_count : INT := 0;
    best_agc : REAL := 0.0;
    best_az : REAL := 0.0;
    best_el : REAL := 0.0;
    bInit : BOOL;
    icount0 : INT := 0;
    icount1 : INT := 0;
    x : REAL := 0.0;
    y : REAL := 0.0;
    dx : REAL := 1.0;
    dy : REAL := 0.0;
    step_len : REAL := 1.0;
    step_count : REAL := 0.0;
    segment_progress : REAL := 0.0;
    move_count : REAL := 1.0;
    state : INT := 0;
    az0 : REAL := 0.0;
    el0 : REAL := 0.0;
    az1 : REAL := 0.0;
    el1 : REAL := 0.0;
    segment_az_step : REAL := 0.0;
    segment_el_step : REAL := 0.0;
    side_repeat : REAL := 0.0;
    icountInit : INT := 0;
  END_VAR

                    
(*==============================================================================
  FB: SpiralScan_1（捕获扫描：螺旋扫描）
  调用者: `SecurityCheck`（段 11），PersistentVars.bSearchType=TRUE 时使用

  与 SpiralScan 区别:
    - 不做矩形格点，而是在网格上按“右→上→左→下”方向逐圈扩展
    - 每一段线性分割为 n_steps 步输出（segment_*_step）
    - 当达到边界条件（az≈4*delta 且 el≈0）或提前锁定即结束

  输出 best_az/best_el:
    - 每拍若 agc 更大，则记录 best_* = -Error（表示需要反向修正误差）
==============================================================================*)
IF NOT enable THEN
    state := 0;
    azimuth := 0.0;
    elevation := 0.0;
    done := FALSE;
	lock_count := 0;
	icount0 := 0;
	segment_progress := 0.0;
	bInit := FALSE;
	best_agc := 0.0;
    best_az := 0.0;
    best_el := 0.0;
	icountInit := 0;
ELSE
    CASE state OF
        // --- 状态0：判断是否已锁定 ---
        0:
			
            
			icountInit := icountInit + 1;
			IF icountInit >= 100 THEN
				icountInit := 101;
				icount0 := icount0 + 1;
				IF locked THEN
					lock_count := lock_count + 1;
				END_IF;
				IF icount0 >= 100 THEN
					IF lock_count >= 10 THEN
						done := TRUE;
						state := 2;   // 提前结束
						lock_count := 0;
					ELSE
						state := 1;   // 转入扫描
						lock_count := 0;
					END_IF;
				END_IF
			END_IF

        // --- 状态1：执行螺旋扫描 ---
        1:
            IF NOT bInit THEN
				x := 0.0; y := 0.0;
				dx := 1.0; dy := 0.0;
				step_len := 1.0;
				step_count := 0.0;
				move_count := 1.0;
				side_repeat := 0.0;
				az0 := 0.0; el0 := 0.0;
				az1 := delta * x;
				el1 := delta * y;
				segment_az_step := (az1 - az0) / n_steps;
				segment_el_step := (el1 - el0) / n_steps;
				segment_progress := 0.0;
				bInit := TRUE;
			ELSE
				
				
				azimuth := az0 + segment_az_step * (segment_progress + 1.0);
				elevation := el0 + segment_el_step * (segment_progress + 1.0);
				segment_progress := segment_progress + 1.0;
				(*
				IF SQRT(azimuth * azimuth + elevation * elevation) > max_radius THEN
						state := 2;
				END_IF
				*)
				
				IF segment_progress >= n_steps THEN
					segment_progress := 0.0;
					az0 := az1;
					el0 := el1;
					// 曼哈顿坐标前进一格
					x := x + dx;
					y := y + dy;
					move_count := move_count + 1.0;
		
					az1 := delta * x;
					el1 := delta * y;
					segment_az_step := (az1 - az0) / n_steps;
					segment_el_step := (el1 - el0) / n_steps;
		
					// 计数并判断是否转弯
					step_count := step_count + 1.0;
					IF step_count >= step_len THEN
						step_count := 0.0;
		
						// 不使用临时变量交换 dx/dy，改为三步法旋转（右→上→左→下）
						IF dx = 1.0 AND dy = 0.0 THEN
							dx := 0.0; dy := 1.0;
						ELSIF dx = 0.0 AND dy = 1.0 THEN
							dx := -1.0; dy := 0.0;
						ELSIF dx = -1.0 AND dy = 0.0 THEN
							dx := 0.0; dy := -1.0;
						ELSIF dx = 0.0 AND dy = -1.0 THEN
							dx := 1.0; dy := 0.0;
						END_IF
		
						side_repeat := side_repeat + 1.0;
						IF side_repeat >= 2.0 THEN
							side_repeat := 0.0;
							step_len := step_len + 1.0;
						END_IF
					END_IF
					
					
				END_IF
				
				IF agc > best_agc THEN
					best_agc := agc;
					best_az := -Azerror;
					best_el := -elError;
				END_IF;
				
				IF ABS(azimuth - 4 * delta) < 1E-6 AND ABS(elevation) < 1E-6 THEN
					state := 3;
				ELSE
					IF locked THEN
					   lock_count := lock_count + 1;
					ELSE
					   lock_count := 0;
					END_IF
					IF lock_count >= 10 THEN
					   done := TRUE;
					   state := 2;   // 提前结束
					   azimuth := best_az;
            		   elevation := best_el;
					END_IF
				END_IF
				
				
			END_IF
        // --- 状态2：提前锁定完成 ---
        2:
            // 保持当前位置即可
            done := TRUE;
			

        // --- 状态3：完成，输出最佳格点 ---
        3:
            azimuth := best_az;
            elevation := best_el;
            done := TRUE;

    END_CASE
	IF state = 3 THEN
		bType := FALSE;
	ELSE
		bType := TRUE;
	END_IF
END_IF;
                  
END_FUNCTION_BLOCK

